KUKA KRL program: f1_Kuka_APT208T02S08.SRC

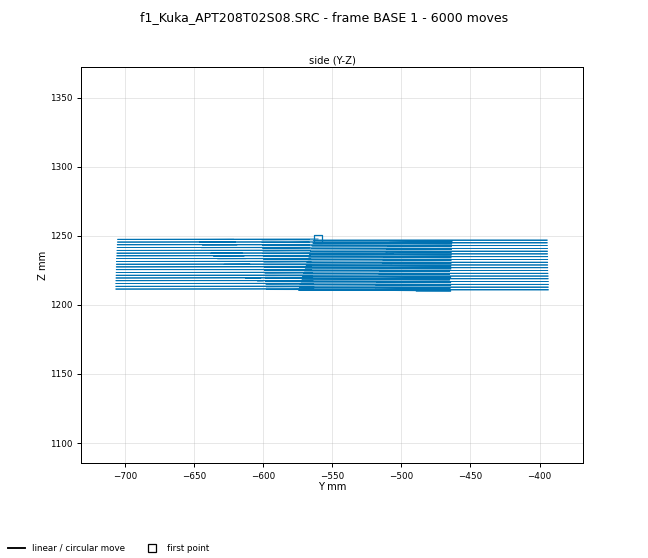
[picture p0: tool path of f1_Kuka_APT208T02S08.SRC in frame BASE 1, 6000 of 6001 moves have a stored position in this frame; points joined in program order, loops and branches not executed]
&ACCESS RVP
&REL 2
&PARAM TEMPLATE = C:\KRC\Roboter\Template\vorgabe
&PARAM EDITMASK = *
DEF f1_Kuka_APT208T02S08()


;FOLD INI;%{PE}%V3.2.0,%MKUKATPBASIS,%CINIT,%VCOMMON,%P
  ;FOLD BAS INI;%{E}%V3.2.0,%MKUKATPBASIS,%CINIT,%VINIT,%P
    GLOBAL INTERRUPT DECL 3 WHEN $STOPMESS==TRUE DO IR_STOPM ( )
    INTERRUPT ON 3
    BAS (#INITMOV,0 )
  ;ENDFOLD (BAS INI)
  ;FOLD USER INI;%{E}%V3.2.0,%MKUKATPUSER,%CINIT,%VINIT,%P
    ;Make your modifications here
  ;ENDFOLD (USER INI)
;ENDFOLD (INI)


;*** Make Null PTP Move
  PTP $pos_act

;*** Auto Load The Correct TOOL Data
  $tool=tool_data[2]

;*** Auto Load The Correct BASE Data
  $base=base_data[1]

  $ADVANCE = 5

;*** Restate Last Velocity
MMPM(30000.0)
SetRPM(8000)
LIN {X -0.044,Y -560.210,Z 1247.711,A 0.000,B 0.000,C 90.000,E1 163.921} C_DIS
LIN {X 0.207,Y -563.468,Z 1247.701,A 0.000,B 0.000,C 90.000,E1 162.236} C_DIS
LIN {X 0.002,Y -567.714,Z 1247.692,A 0.000,B 0.000,C 90.000,E1 160.604} C_DIS
LIN {X 0.261,Y -572.378,Z 1247.685,A 0.000,B 0.000,C 90.000,E1 159.209} C_DIS
LIN {X -0.101,Y -576.704,Z 1247.679,A 0.000,B 0.000,C 90.000,E1 158.156} C_DIS
LIN {X 0.147,Y -589.999,Z 1247.663,A 0.000,B 0.000,C 90.000,E1 155.305} C_DIS
LIN {X 0.135,Y -597.371,Z 1247.655,A 0.000,B 0.000,C 90.000,E1 153.845} C_DIS
LIN {X 0.131,Y -601.919,Z 1247.650,A 0.000,B 0.000,C 90.000,E1 152.922} C_DIS
LIN {X 0.032,Y -603.823,Z 1247.647,A 0.000,B 0.000,C 90.000,E1 152.538} C_DIS
LIN {X -0.143,Y -607.711,Z 1247.643,A 0.000,B 0.000,C 90.000,E1 151.769} C_DIS
LIN {X 0.008,Y -611.290,Z 1247.639,A 0.000,B 0.000,C 90.000,E1 150.973} C_DIS
LIN {X 0.120,Y -618.388,Z 1247.630,A 0.000,B 0.000,C 90.000,E1 149.410} C_DIS
LIN {X 0.147,Y -625.351,Z 1247.622,A 0.000,B 0.000,C 90.000,E1 147.867} C_DIS
LIN {X -0.054,Y -628.614,Z 1247.617,A 0.000,B 0.000,C 90.000,E1 147.120} C_DIS
LIN {X -0.384,Y -633.789,Z 1247.610,A 0.000,B 0.000,C 90.000,E1 145.881} C_DIS
LIN {X -0.147,Y -636.719,Z 1247.606,A 0.000,B 0.000,C 90.000,E1 145.102} C_DIS
LIN {X 0.026,Y -641.252,Z 1247.599,A 0.000,B 0.000,C 90.000,E1 143.829} C_DIS
LIN {X 0.272,Y -645.228,Z 1247.592,A 0.000,B 0.000,C 90.000,E1 142.557} C_DIS
LIN {X -0.366,Y -648.122,Z 1247.587,A 0.000,B 0.000,C 90.000,E1 141.618} C_DIS
LIN {X -0.126,Y -651.565,Z 1247.580,A 0.000,B 0.000,C 90.000,E1 140.356} C_DIS
LIN {X 0.124,Y -655.386,Z 1247.572,A 0.000,B 0.000,C 90.000,E1 138.852} C_DIS
LIN {X 0.020,Y -657.887,Z 1247.566,A 0.000,B 0.000,C 90.000,E1 137.877} C_DIS
LIN {X 0.341,Y -661.423,Z 1247.558,A 0.000,B 0.000,C 90.000,E1 136.377} C_DIS
LIN {X 0.254,Y -667.065,Z 1247.546,A 0.000,B 0.000,C 90.000,E1 134.190} C_DIS
LIN {X -0.167,Y -671.614,Z 1247.536,A 0.000,B 0.000,C 90.000,E1 132.528} C_DIS
LIN {X -0.020,Y -675.508,Z 1247.528,A 0.000,B 0.000,C 90.000,E1 131.067} C_DIS
LIN {X 0.168,Y -678.705,Z 1247.521,A 0.000,B 0.000,C 90.000,E1 129.850} C_DIS
LIN {X 0.172,Y -683.657,Z 1247.511,A 0.000,B 0.000,C 90.000,E1 127.935} C_DIS
LIN {X 0.214,Y -687.311,Z 1247.503,A 0.000,B 0.000,C 90.000,E1 126.503} C_DIS
LIN {X -0.308,Y -689.569,Z 1247.498,A 0.000,B 0.000,C 90.000,E1 125.598} C_DIS
LIN {X -0.197,Y -692.243,Z 1247.491,A 0.000,B 0.000,C 90.000,E1 124.405} C_DIS
LIN {X -0.081,Y -694.262,Z 1247.486,A 0.000,B 0.000,C 90.000,E1 123.452} C_DIS
LIN {X 0.093,Y -696.685,Z 1247.479,A 0.000,B 0.000,C 90.000,E1 122.260} C_DIS
LIN {X 0.151,Y -698.904,Z 1247.473,A 0.000,B 0.000,C 90.000,E1 121.082} C_DIS
LIN {X 0.008,Y -701.036,Z 1247.466,A 0.000,B 0.000,C 90.000,E1 119.922} C_DIS
LIN {X 0.209,Y -702.176,Z 1247.462,A 0.000,B 0.000,C 90.000,E1 119.205} C_DIS
LIN {X 0.084,Y -703.477,Z 1247.457,A 0.000,B 0.000,C 90.000,E1 118.281} C_DIS
LIN {X -0.359,Y -704.484,Z 1247.452,A 0.000,B 0.000,C 90.000,E1 117.385} C_DIS
LIN {X -0.127,Y -705.034,Z 1247.448,A 0.000,B 0.000,C 90.000,E1 116.668} C_DIS
LIN {X -0.206,Y -705.331,Z 1247.444,A 0.000,B 0.000,C 90.000,E1 115.976} C_DIS
LIN {X 0.373,Y -705.331,Z 1247.442,A 0.000,B 0.000,C 90.000,E1 115.463} C_DIS
LIN {X 0.013,Y -705.151,Z 1247.439,A 0.000,B 0.000,C 90.000,E1 115.027} C_DIS
LIN {X -0.052,Y -704.772,Z 1247.437,A 0.000,B 0.000,C 90.000,E1 114.567} C_DIS
LIN {X 0.229,Y -703.978,Z 1247.434,A 0.000,B 0.000,C 90.000,E1 114.079} C_DIS
LIN {X -0.131,Y -703.306,Z 1247.433,A 0.000,B 0.000,C 90.000,E1 113.875} C_DIS
LIN {X 0.144,Y -701.285,Z 1247.430,A 0.000,B 0.000,C 90.000,E1 113.387} C_DIS
LIN {X 0.280,Y -700.576,Z 1247.429,A 0.000,B 0.000,C 90.000,E1 113.259} C_DIS
LIN {X -0.106,Y -696.209,Z 1247.427,A 0.000,B 0.000,C 90.000,E1 112.823} C_DIS
LIN {X 0.023,Y -694.918,Z 1247.426,A 0.000,B 0.000,C 90.000,E1 112.695} C_DIS
LIN {X -0.059,Y -692.962,Z 1247.426,A 0.000,B 0.000,C 90.000,E1 112.589} C_DIS
LIN {X 0.208,Y -686.106,Z 1247.424,A 0.000,B 0.000,C 90.000,E1 112.333} C_DIS
LIN {X -0.047,Y -684.944,Z 1247.424,A 0.000,B 0.000,C 90.000,E1 112.333} C_DIS
LIN {X -0.092,Y -677.360,Z 1247.424,A 0.000,B 0.000,C 90.000,E1 112.259} C_DIS
LIN {X -0.131,Y -625.323,Z 1247.424,A 0.000,B 0.000,C 90.000,E1 112.259} C_DIS
LIN {X -0.005,Y -624.460,Z 1247.423,A 0.000,B 0.000,C 90.000,E1 112.206} C_DIS
LIN {X -0.259,Y -621.696,Z 1247.422,A 0.000,B 0.000,C 90.000,E1 112.025} C_DIS
LIN {X -0.295,Y -621.657,Z 1247.422,A 0.000,B 0.000,C 90.000,E1 112.025} C_DIS
LIN {X -0.018,Y -621.126,Z 1247.422,A 0.000,B 0.000,C 90.000,E1 111.897} C_DIS
LIN {X -0.061,Y -621.110,Z 1247.422,A 0.000,B 0.000,C 90.000,E1 111.897} C_DIS
LIN {X -0.234,Y -621.700,Z 1247.420,A 0.000,B 0.000,C 90.000,E1 111.589} C_DIS
LIN {X 0.091,Y -625.646,Z 1247.416,A 0.000,B 0.000,C 90.000,E1 110.791} C_DIS
LIN {X -0.347,Y -630.528,Z 1247.411,A 0.000,B 0.000,C 90.000,E1 109.939} C_DIS
LIN {X 0.056,Y -633.087,Z 1247.408,A 0.000,B 0.000,C 90.000,E1 109.396} C_DIS
LIN {X 0.311,Y -637.748,Z 1247.402,A 0.000,B 0.000,C 90.000,E1 108.362} C_DIS
LIN {X 0.156,Y -646.024,Z 1247.392,A 0.000,B 0.000,C 90.000,E1 106.622} C_DIS
LIN {X 0.043,Y -648.319,Z 1247.390,A 0.000,B 0.000,C 90.000,E1 106.134} C_DIS
LIN {X 0.257,Y -651.410,Z 1247.386,A 0.000,B 0.000,C 90.000,E1 105.371} C_DIS
LIN {X 0.003,Y -653.197,Z 1247.383,A 0.000,B 0.000,C 90.000,E1 104.898} C_DIS
LIN {X -0.197,Y -655.418,Z 1247.379,A 0.000,B 0.000,C 90.000,E1 104.175} C_DIS
LIN {X 0.208,Y -656.599,Z 1247.376,A 0.000,B 0.000,C 90.000,E1 103.647} C_DIS
LIN {X -0.126,Y -657.857,Z 1247.372,A 0.000,B 0.000,C 90.000,E1 102.939} C_DIS
LIN {X 0.298,Y -658.390,Z 1247.369,A 0.000,B 0.000,C 90.000,E1 102.411} C_DIS
LIN {X -0.054,Y -658.521,Z 1247.366,A 0.000,B 0.000,C 90.000,E1 101.951} C_DIS
LIN {X 0.273,Y -658.185,Z 1247.362,A 0.000,B 0.000,C 90.000,E1 101.186} C_DIS
LIN {X 0.054,Y -657.548,Z 1247.360,A 0.000,B 0.000,C 90.000,E1 100.715} C_DIS
LIN {X -0.290,Y -656.626,Z 1247.357,A 0.000,B 0.000,C 90.000,E1 100.254} C_DIS
LIN {X 0.124,Y -655.438,Z 1247.354,A 0.000,B 0.000,C 90.000,E1 99.726} C_DIS
LIN {X -0.105,Y -654.766,Z 1247.353,A 0.000,B 0.000,C 90.000,E1 99.500} C_DIS
LIN {X 0.293,Y -653.009,Z 1247.350,A 0.000,B 0.000,C 90.000,E1 98.973} C_DIS
LIN {X -0.070,Y -650.852,Z 1247.347,A 0.000,B 0.000,C 90.000,E1 98.511} C_DIS
LIN {X 0.171,Y -647.758,Z 1247.344,A 0.000,B 0.000,C 90.000,E1 97.871} C_DIS
LIN {X 0.294,Y -644.050,Z 1247.340,A 0.000,B 0.000,C 90.000,E1 97.239} C_DIS
LIN {X -0.248,Y -639.738,Z 1247.337,A 0.000,B 0.000,C 90.000,E1 96.663} C_DIS
LIN {X 0.077,Y -636.974,Z 1247.335,A 0.000,B 0.000,C 90.000,E1 96.258} C_DIS
LIN {X 0.143,Y -631.622,Z 1247.331,A 0.000,B 0.000,C 90.000,E1 95.625} C_DIS
LIN {X -0.307,Y -626.824,Z 1247.329,A 0.000,B 0.000,C 90.000,E1 95.163} C_DIS
LIN {X -0.030,Y -620.264,Z 1247.325,A 0.000,B 0.000,C 90.000,E1 94.531} C_DIS
LIN {X -0.028,Y -614.926,Z 1247.323,A 0.000,B 0.000,C 90.000,E1 94.073} C_DIS
LIN {X 0.146,Y -609.256,Z 1247.320,A 0.000,B 0.000,C 90.000,E1 93.612} C_DIS
LIN {X 0.021,Y -601.636,Z 1247.317,A 0.000,B 0.000,C 90.000,E1 93.094} C_DIS
LIN {X 0.005,Y -595.380,Z 1247.315,A 0.000,B 0.000,C 90.000,E1 92.694} C_DIS
LIN {X 0.222,Y -588.941,Z 1247.313,A 0.000,B 0.000,C 90.000,E1 92.293} C_DIS
LIN {X 0.267,Y -582.256,Z 1247.311,A 0.000,B 0.000,C 90.000,E1 91.949} C_DIS
LIN {X 0.028,Y -571.609,Z 1247.309,A 0.000,B 0.000,C 90.000,E1 91.547} C_DIS
LIN {X -0.094,Y -570.151,Z 1247.308,A 0.000,B 0.000,C 90.000,E1 91.489} C_DIS
LIN {X -0.132,Y -568.129,Z 1247.308,A 0.000,B 0.000,C 90.000,E1 91.375} C_DIS
LIN {X -0.189,Y -568.057,Z 1247.308,A 0.000,B 0.000,C 90.000,E1 91.375} C_DIS
LIN {X 0.032,Y -566.808,Z 1247.306,A 0.000,B 0.000,C 90.000,E1 91.088} C_DIS
LIN {X -0.010,Y -566.801,Z 1247.306,A 0.000,B 0.000,C 90.000,E1 91.088} C_DIS
LIN {X 0.198,Y -566.625,Z 1247.304,A 0.000,B 0.000,C 90.000,E1 90.630} C_DIS
LIN {X -0.016,Y -567.066,Z 1247.299,A 0.000,B 0.000,C 90.000,E1 89.828} C_DIS
LIN {X 0.153,Y -568.269,Z 1247.290,A 0.000,B 0.000,C 90.000,E1 88.165} C_DIS
LIN {X 0.024,Y -570.020,Z 1247.278,A 0.000,B 0.000,C 90.000,E1 85.988} C_DIS
LIN {X -0.118,Y -571.911,Z 1247.267,A 0.000,B 0.000,C 90.000,E1 84.090} C_DIS
LIN {X 0.298,Y -573.564,Z 1247.258,A 0.000,B 0.000,C 90.000,E1 82.413} C_DIS
LIN {X -0.014,Y -574.966,Z 1247.250,A 0.000,B 0.000,C 90.000,E1 81.084} C_DIS
LIN {X 0.143,Y -575.994,Z 1247.245,A 0.000,B 0.000,C 90.000,E1 79.982} C_DIS
LIN {X 0.064,Y -577.006,Z 1247.237,A 0.000,B 0.000,C 90.000,E1 78.634} C_DIS
LIN {X 0.014,Y -577.979,Z 1247.229,A 0.000,B 0.000,C 90.000,E1 77.285} C_DIS
LIN {X 0.102,Y -578.547,Z 1247.225,A 0.000,B 0.000,C 90.000,E1 76.464} C_DIS
LIN {X 0.211,Y -579.429,Z 1247.217,A 0.000,B 0.000,C 90.000,E1 75.102} C_DIS
LIN {X -0.011,Y -580.339,Z 1247.208,A 0.000,B 0.000,C 90.000,E1 73.504} C_DIS
LIN {X 0.115,Y -581.232,Z 1247.199,A 0.000,B 0.000,C 90.000,E1 71.873} C_DIS
LIN {X -0.131,Y -582.131,Z 1247.192,A 0.000,B 0.000,C 90.000,E1 70.550} C_DIS
LIN {X 0.140,Y -583.605,Z 1247.178,A 0.000,B 0.000,C 90.000,E1 68.103} C_DIS
LIN {X -0.050,Y -585.213,Z 1247.167,A 0.000,B 0.000,C 90.000,E1 65.973} C_DIS
LIN {X -0.250,Y -586.167,Z 1247.161,A 0.000,B 0.000,C 90.000,E1 64.921} C_DIS
LIN {X 0.016,Y -588.286,Z 1247.147,A 0.000,B 0.000,C 90.000,E1 62.487} C_DIS
LIN {X 0.143,Y -589.936,Z 1247.138,A 0.000,B 0.000,C 90.000,E1 60.873} C_DIS
LIN {X 0.181,Y -591.324,Z 1247.131,A 0.000,B 0.000,C 90.000,E1 59.537} C_DIS
LIN {X 0.249,Y -592.705,Z 1247.124,A 0.000,B 0.000,C 90.000,E1 58.201} C_DIS
LIN {X -0.166,Y -593.989,Z 1247.116,A 0.000,B 0.000,C 90.000,E1 56.914} C_DIS
LIN {X -0.010,Y -595.441,Z 1247.107,A 0.000,B 0.000,C 90.000,E1 55.308} C_DIS
LIN {X 0.179,Y -596.833,Z 1247.099,A 0.000,B 0.000,C 90.000,E1 53.703} C_DIS
LIN {X -0.336,Y -598.277,Z 1247.088,A 0.000,B 0.000,C 90.000,E1 51.904} C_DIS
LIN {X 0.142,Y -599.069,Z 1247.082,A 0.000,B 0.000,C 90.000,E1 50.803} C_DIS
LIN {X 0.189,Y -599.846,Z 1247.074,A 0.000,B 0.000,C 90.000,E1 49.218} C_DIS
LIN {X 0.229,Y -600.315,Z 1247.068,A 0.000,B 0.000,C 90.000,E1 48.162} C_DIS
LIN {X 0.037,Y -600.654,Z 1247.063,A 0.000,B 0.000,C 90.000,E1 47.391} C_DIS
LIN {X 0.068,Y -600.929,Z 1247.055,A 0.000,B 0.000,C 90.000,E1 45.810} C_DIS
LIN {X 0.090,Y -600.994,Z 1247.049,A 0.000,B 0.000,C 90.000,E1 44.757} C_DIS
LIN {X 0.111,Y -600.833,Z 1247.043,A 0.000,B 0.000,C 90.000,E1 43.704} C_DIS
LIN {X -0.055,Y -600.482,Z 1247.036,A 0.000,B 0.000,C 90.000,E1 42.405} C_DIS
LIN {X -0.040,Y -599.793,Z 1247.027,A 0.000,B 0.000,C 90.000,E1 40.825} C_DIS
LIN {X 0.229,Y -599.080,Z 1247.020,A 0.000,B 0.000,C 90.000,E1 39.483} C_DIS
LIN {X -0.127,Y -598.295,Z 1247.014,A 0.000,B 0.000,C 90.000,E1 38.463} C_DIS
LIN {X 0.111,Y -597.624,Z 1247.009,A 0.000,B 0.000,C 90.000,E1 37.649} C_DIS
LIN {X 0.211,Y -596.519,Z 1247.003,A 0.000,B 0.000,C 90.000,E1 36.583} C_DIS
LIN {X 0.296,Y -595.048,Z 1246.998,A 0.000,B 0.000,C 90.000,E1 35.518} C_DIS
LIN {X 0.136,Y -593.782,Z 1246.993,A 0.000,B 0.000,C 90.000,E1 34.739} C_DIS
LIN {X -0.159,Y -591.802,Z 1246.987,A 0.000,B 0.000,C 90.000,E1 33.706} C_DIS
LIN {X 0.135,Y -590.025,Z 1246.983,A 0.000,B 0.000,C 90.000,E1 32.880} C_DIS
LIN {X 0.214,Y -588.683,Z 1246.980,A 0.000,B 0.000,C 90.000,E1 32.339} C_DIS
LIN {X 0.161,Y -586.395,Z 1246.975,A 0.000,B 0.000,C 90.000,E1 31.544} C_DIS
LIN {X 0.091,Y -583.801,Z 1246.971,A 0.000,B 0.000,C 90.000,E1 30.747} C_DIS
LIN {X -0.006,Y -580.713,Z 1246.966,A 0.000,B 0.000,C 90.000,E1 29.951} C_DIS
LIN {X 0.008,Y -578.463,Z 1246.964,A 0.000,B 0.000,C 90.000,E1 29.411} C_DIS
LIN {X 0.000,Y -575.979,Z 1246.960,A 0.000,B 0.000,C 90.000,E1 28.871} C_DIS
LIN {X 0.228,Y -571.161,Z 1246.955,A 0.000,B 0.000,C 90.000,E1 27.897} C_DIS
LIN {X -0.280,Y -566.486,Z 1246.951,A 0.000,B 0.000,C 90.000,E1 27.129} C_DIS
LIN {X 0.116,Y -563.139,Z 1246.948,A 0.000,B 0.000,C 90.000,E1 26.539} C_DIS
LIN {X 0.233,Y -559.571,Z 1246.944,A 0.000,B 0.000,C 90.000,E1 25.976} C_DIS
LIN {X -0.175,Y -555.773,Z 1246.941,A 0.000,B 0.000,C 90.000,E1 25.463} C_DIS
LIN {X -0.105,Y -551.668,Z 1246.938,A 0.000,B 0.000,C 90.000,E1 24.899} C_DIS
LIN {X 0.196,Y -545.099,Z 1246.934,A 0.000,B 0.000,C 90.000,E1 24.027} C_DIS
LIN {X 0.123,Y -539.158,Z 1246.930,A 0.000,B 0.000,C 90.000,E1 23.334} C_DIS
LIN {X -0.172,Y -531.578,Z 1246.925,A 0.000,B 0.000,C 90.000,E1 22.514} C_DIS
LIN {X 0.065,Y -524.997,Z 1246.921,A 0.000,B 0.000,C 90.000,E1 21.791} C_DIS
LIN {X -0.124,Y -515.656,Z 1246.916,A 0.000,B 0.000,C 90.000,E1 20.844} C_DIS
LIN {X 0.061,Y -507.377,Z 1246.911,A 0.000,B 0.000,C 90.000,E1 19.993} C_DIS
LIN {X -0.230,Y -497.632,Z 1246.906,A 0.000,B 0.000,C 90.000,E1 19.087} C_DIS
LIN {X -0.071,Y -487.541,Z 1246.901,A 0.000,B 0.000,C 90.000,E1 18.127} C_DIS
LIN {X -0.049,Y -478.666,Z 1246.896,A 0.000,B 0.000,C 90.000,E1 17.330} C_DIS
LIN {X -0.150,Y -462.368,Z 1246.888,A 0.000,B 0.000,C 90.000,E1 15.898} C_DIS
LIN {X -0.017,Y -446.234,Z 1246.880,A 0.000,B 0.000,C 90.000,E1 14.411} C_DIS
LIN {X 0.099,Y -424.423,Z 1246.868,A 0.000,B 0.000,C 90.000,E1 12.243} C_DIS
LIN {X -0.111,Y -405.887,Z 1246.857,A 0.000,B 0.000,C 90.000,E1 10.254} C_DIS
LIN {X -0.165,Y -401.633,Z 1246.854,A 0.000,B 0.000,C 90.000,E1 9.782} C_DIS
LIN {X 0.209,Y -396.128,Z 1246.850,A 0.000,B 0.000,C 90.000,E1 8.973} C_DIS
LIN {X 0.139,Y -394.399,Z 1246.848,A 0.000,B 0.000,C 90.000,E1 8.624} C_DIS
LIN {X 0.103,Y -394.392,Z 1246.848,A 0.000,B 0.000,C 90.000,E1 8.624} C_DIS
LIN {X -0.056,Y -394.298,Z 1246.848,A 0.000,B 0.000,C 90.000,E1 8.568} C_DIS
LIN {X -0.092,Y -394.300,Z 1246.848,A 0.000,B 0.000,C 90.000,E1 8.568} C_DIS
LIN {X -0.043,Y -396.382,Z 1246.845,A 0.000,B 0.000,C 90.000,E1 8.106} C_DIS
LIN {X 0.065,Y -400.030,Z 1246.843,A 0.000,B 0.000,C 90.000,E1 7.701} C_DIS
LIN {X -0.161,Y -405.750,Z 1246.840,A 0.000,B 0.000,C 90.000,E1 7.296} C_DIS
LIN {X -0.113,Y -412.470,Z 1246.838,A 0.000,B 0.000,C 90.000,E1 6.834} C_DIS
LIN {X -0.049,Y -423.583,Z 1246.833,A 0.000,B 0.000,C 90.000,E1 6.030} C_DIS
LIN {X -0.118,Y -431.436,Z 1246.830,A 0.000,B 0.000,C 90.000,E1 5.448} C_DIS
LIN {X -0.078,Y -440.778,Z 1246.826,A 0.000,B 0.000,C 90.000,E1 4.702} C_DIS
LIN {X -0.019,Y -448.647,Z 1246.823,A 0.000,B 0.000,C 90.000,E1 4.073} C_DIS
LIN {X -0.185,Y -459.503,Z 1246.818,A 0.000,B 0.000,C 90.000,E1 3.212} C_DIS
LIN {X -0.227,Y -467.080,Z 1246.814,A 0.000,B 0.000,C 90.000,E1 2.579} C_DIS
LIN {X 0.174,Y -472.961,Z 1246.811,A 0.000,B 0.000,C 90.000,E1 2.007} C_DIS
LIN {X -0.051,Y -478.704,Z 1246.808,A 0.000,B 0.000,C 90.000,E1 1.489} C_DIS
LIN {X -0.207,Y -485.431,Z 1246.804,A 0.000,B 0.000,C 90.000,E1 0.802} C_DIS
LIN {X 0.000,Y -492.261,Z 1246.800,A 0.000,B 0.000,C 90.000,E1 360.000} C_DIS
LIN {X 0.038,Y -496.537,Z 1246.797,A 0.000,B 0.000,C 90.000,E1 359.484} C_DIS
LIN {X 0.141,Y -503.300,Z 1246.792,A 0.000,B 0.000,C 90.000,E1 358.568} C_DIS
LIN {X -0.071,Y -507.579,Z 1246.789,A 0.000,B 0.000,C 90.000,E1 357.993} C_DIS
LIN {X -0.058,Y -512.453,Z 1246.785,A 0.000,B 0.000,C 90.000,E1 357.249} C_DIS
LIN {X 0.021,Y -517.080,Z 1246.781,A 0.000,B 0.000,C 90.000,E1 356.502} C_DIS
LIN {X -0.081,Y -520.544,Z 1246.777,A 0.000,B 0.000,C 90.000,E1 355.927} C_DIS
LIN {X 0.080,Y -524.508,Z 1246.773,A 0.000,B 0.000,C 90.000,E1 355.179} C_DIS
LIN {X 0.279,Y -528.131,Z 1246.769,A 0.000,B 0.000,C 90.000,E1 354.432} C_DIS
LIN {X 0.261,Y -530.849,Z 1246.766,A 0.000,B 0.000,C 90.000,E1 353.856} C_DIS
LIN {X 0.262,Y -533.398,Z 1246.763,A 0.000,B 0.000,C 90.000,E1 353.280} C_DIS
LIN {X -0.254,Y -535.770,Z 1246.760,A 0.000,B 0.000,C 90.000,E1 352.761} C_DIS
LIN {X -0.170,Y -538.958,Z 1246.755,A 0.000,B 0.000,C 90.000,E1 351.894} C_DIS
LIN {X 0.021,Y -542.828,Z 1246.749,A 0.000,B 0.000,C 90.000,E1 350.735} C_DIS
LIN {X 0.270,Y -545.377,Z 1246.744,A 0.000,B 0.000,C 90.000,E1 349.859} C_DIS
LIN {X 0.012,Y -548.535,Z 1246.738,A 0.000,B 0.000,C 90.000,E1 348.757} C_DIS
LIN {X -0.212,Y -550.682,Z 1246.733,A 0.000,B 0.000,C 90.000,E1 347.937} C_DIS
LIN {X -0.299,Y -553.228,Z 1246.727,A 0.000,B 0.000,C 90.000,E1 346.825} C_DIS
LIN {X -0.221,Y -555.597,Z 1246.720,A 0.000,B 0.000,C 90.000,E1 345.700} C_DIS
LIN {X -0.237,Y -557.140,Z 1246.716,A 0.000,B 0.000,C 90.000,E1 344.866} C_DIS
LIN {X -0.100,Y -559.042,Z 1246.710,A 0.000,B 0.000,C 90.000,E1 343.740} C_DIS
LIN {X -0.080,Y -560.216,Z 1246.705,A 0.000,B 0.000,C 90.000,E1 342.906} C_DIS
LIN {X -0.278,Y -561.613,Z 1246.699,A 0.000,B 0.000,C 90.000,E1 341.819} C_DIS
LIN {X 0.074,Y -562.633,Z 1246.693,A 0.000,B 0.000,C 90.000,E1 340.678} C_DIS
LIN {X -0.225,Y -563.146,Z 1246.688,A 0.000,B 0.000,C 90.000,E1 339.880} C_DIS
LIN {X 0.012,Y -563.378,Z 1246.684,A 0.000,B 0.000,C 90.000,E1 339.028} C_DIS
LIN {X 0.131,Y -563.407,Z 1246.681,A 0.000,B 0.000,C 90.000,E1 338.465} C_DIS
LIN {X -0.155,Y -563.100,Z 1246.676,A 0.000,B 0.000,C 90.000,E1 337.667} C_DIS
LIN {X -0.032,Y -562.690,Z 1246.673,A 0.000,B 0.000,C 90.000,E1 337.102} C_DIS
LIN {X -0.018,Y -561.489,Z 1246.667,A 0.000,B 0.000,C 90.000,E1 335.997} C_DIS
LIN {X 0.092,Y -560.672,Z 1246.664,A 0.000,B 0.000,C 90.000,E1 335.433} C_DIS
LIN {X 0.232,Y -559.167,Z 1246.659,A 0.000,B 0.000,C 90.000,E1 334.588} C_DIS
LIN {X -0.299,Y -556.141,Z 1246.651,A 0.000,B 0.000,C 90.000,E1 333.256} C_DIS
LIN {X -0.193,Y -553.609,Z 1246.647,A 0.000,B 0.000,C 90.000,E1 332.410} C_DIS
LIN {X -0.113,Y -550.710,Z 1246.642,A 0.000,B 0.000,C 90.000,E1 331.563} C_DIS
LIN {X 0.054,Y -547.836,Z 1246.638,A 0.000,B 0.000,C 90.000,E1 330.845} C_DIS
LIN {X 0.189,Y -544.503,Z 1246.634,A 0.000,B 0.000,C 90.000,E1 330.127} C_DIS
LIN {X -0.180,Y -540.698,Z 1246.630,A 0.000,B 0.000,C 90.000,E1 329.459} C_DIS
LIN {X 0.023,Y -535.345,Z 1246.625,A 0.000,B 0.000,C 90.000,E1 328.584} C_DIS
LIN {X 0.013,Y -528.671,Z 1246.620,A 0.000,B 0.000,C 90.000,E1 327.582} C_DIS
LIN {X 0.073,Y -522.477,Z 1246.615,A 0.000,B 0.000,C 90.000,E1 326.707} C_DIS
LIN {X -0.080,Y -516.644,Z 1246.610,A 0.000,B 0.000,C 90.000,E1 325.881} C_DIS
LIN {X 0.194,Y -513.232,Z 1246.607,A 0.000,B 0.000,C 90.000,E1 325.308} C_DIS
LIN {X 0.218,Y -510.256,Z 1246.604,A 0.000,B 0.000,C 90.000,E1 324.769} C_DIS
LIN {X -0.293,Y -507.821,Z 1246.601,A 0.000,B 0.000,C 90.000,E1 324.196} C_DIS
LIN {X 0.126,Y -506.615,Z 1246.599,A 0.000,B 0.000,C 90.000,E1 323.703} C_DIS
LIN {X -0.173,Y -504.975,Z 1246.594,A 0.000,B 0.000,C 90.000,E1 322.844} C_DIS
LIN {X 0.217,Y -504.261,Z 1246.589,A 0.000,B 0.000,C 90.000,E1 321.904} C_DIS
LIN {X -0.112,Y -504.155,Z 1246.584,A 0.000,B 0.000,C 90.000,E1 321.045} C_DIS
LIN {X 0.179,Y -504.992,Z 1246.569,A 0.000,B 0.000,C 90.000,E1 318.324} C_DIS
LIN {X -0.015,Y -505.613,Z 1246.557,A 0.000,B 0.000,C 90.000,E1 316.257} C_DIS
LIN {X -0.165,Y -505.927,Z 1246.550,A 0.000,B 0.000,C 90.000,E1 315.081} C_DIS
LIN {X 0.153,Y -506.372,Z 1246.540,A 0.000,B 0.000,C 90.000,E1 313.257} C_DIS
LIN {X 0.016,Y -506.745,Z 1246.534,A 0.000,B 0.000,C 90.000,E1 312.081} C_DIS
LIN {X -0.002,Y -507.285,Z 1246.524,A 0.000,B 0.000,C 90.000,E1 310.297} C_DIS
LIN {X -0.083,Y -507.528,Z 1246.517,A 0.000,B 0.000,C 90.000,E1 309.116} C_DIS
LIN {X 0.050,Y -508.042,Z 1246.507,A 0.000,B 0.000,C 90.000,E1 307.317} C_DIS
LIN {X -0.026,Y -508.356,Z 1246.501,A 0.000,B 0.000,C 90.000,E1 306.137} C_DIS
LIN {X -0.090,Y -508.583,Z 1246.493,A 0.000,B 0.000,C 90.000,E1 304.659} C_DIS
LIN {X -0.013,Y -508.797,Z 1246.484,A 0.000,B 0.000,C 90.000,E1 303.166} C_DIS
LIN {X 0.075,Y -508.907,Z 1246.476,A 0.000,B 0.000,C 90.000,E1 301.671} C_DIS
LIN {X -0.134,Y -508.877,Z 1246.464,A 0.000,B 0.000,C 90.000,E1 299.617} C_DIS
LIN {X 0.046,Y -508.833,Z 1246.458,A 0.000,B 0.000,C 90.000,E1 298.409} C_DIS
LIN {X 0.058,Y -508.718,Z 1246.450,A 0.000,B 0.000,C 90.000,E1 296.924} C_DIS
LIN {X -0.111,Y -508.723,Z 1246.437,A 0.000,B 0.000,C 90.000,E1 294.567} C_DIS
LIN {X 0.089,Y -508.797,Z 1246.433,A 0.000,B 0.000,C 90.000,E1 293.951} C_DIS
LIN {X 0.136,Y -508.606,Z 1246.425,A 0.000,B 0.000,C 90.000,E1 292.461} C_DIS
LIN {X -0.027,Y -508.324,Z 1246.420,A 0.000,B 0.000,C 90.000,E1 291.589} C_DIS
LIN {X -0.179,Y -507.655,Z 1246.412,A 0.000,B 0.000,C 90.000,E1 290.120} C_DIS
LIN {X 0.156,Y -506.724,Z 1246.400,A 0.000,B 0.000,C 90.000,E1 288.000} C_DIS
LIN {X 0.204,Y -506.342,Z 1246.394,A 0.000,B 0.000,C 90.000,E1 286.804} C_DIS
LIN {X 0.188,Y -505.727,Z 1246.385,A 0.000,B 0.000,C 90.000,E1 285.315} C_DIS
LIN {X 0.158,Y -504.856,Z 1246.377,A 0.000,B 0.000,C 90.000,E1 283.828} C_DIS
LIN {X -0.080,Y -503.616,Z 1246.367,A 0.000,B 0.000,C 90.000,E1 282.063} C_DIS
LIN {X 0.043,Y -502.285,Z 1246.357,A 0.000,B 0.000,C 90.000,E1 280.254} C_DIS
LIN {X 0.121,Y -501.261,Z 1246.349,A 0.000,B 0.000,C 90.000,E1 278.746} C_DIS
LIN {X -0.259,Y -499.624,Z 1246.334,A 0.000,B 0.000,C 90.000,E1 276.087} C_DIS
LIN {X 0.198,Y -498.885,Z 1246.325,A 0.000,B 0.000,C 90.000,E1 274.531} C_DIS
LIN {X -0.041,Y -497.836,Z 1246.315,A 0.000,B 0.000,C 90.000,E1 272.751} C_DIS
LIN {X -0.058,Y -496.883,Z 1246.309,A 0.000,B 0.000,C 90.000,E1 271.547} C_DIS
LIN {X -0.157,Y -495.147,Z 1246.295,A 0.000,B 0.000,C 90.000,E1 269.141} C_DIS
LIN {X -0.008,Y -493.925,Z 1246.285,A 0.000,B 0.000,C 90.000,E1 267.306} C_DIS
LIN {X -0.155,Y -493.819,Z 1246.283,A 0.000,B 0.000,C 90.000,E1 267.020} C_DIS
LIN {X -0.200,Y -493.064,Z 1246.277,A 0.000,B 0.000,C 90.000,E1 265.812} C_DIS
LIN {X 0.086,Y -492.259,Z 1246.268,A 0.000,B 0.000,C 90.000,E1 264.261} C_DIS
LIN {X -0.090,Y -491.179,Z 1246.260,A 0.000,B 0.000,C 90.000,E1 262.761} C_DIS
LIN {X 0.264,Y -489.818,Z 1246.251,A 0.000,B 0.000,C 90.000,E1 261.197} C_DIS
LIN {X -0.241,Y -487.525,Z 1246.238,A 0.000,B 0.000,C 90.000,E1 258.814} C_DIS
LIN {X 0.098,Y -486.156,Z 1246.228,A 0.000,B 0.000,C 90.000,E1 256.937} C_DIS
LIN {X 0.051,Y -485.013,Z 1246.217,A 0.000,B 0.000,C 90.000,E1 255.102} C_DIS
LIN {X 0.110,Y -484.152,Z 1246.209,A 0.000,B 0.000,C 90.000,E1 253.559} C_DIS
LIN {X 0.134,Y -482.924,Z 1246.197,A 0.000,B 0.000,C 90.000,E1 251.402} C_DIS
LIN {X -0.022,Y -481.965,Z 1246.187,A 0.000,B 0.000,C 90.000,E1 249.571} C_DIS
LIN {X -0.020,Y -481.180,Z 1246.178,A 0.000,B 0.000,C 90.000,E1 248.028} C_DIS
LIN {X -0.043,Y -480.072,Z 1246.168,A 0.000,B 0.000,C 90.000,E1 246.177} C_DIS
LIN {X 0.098,Y -478.960,Z 1246.159,A 0.000,B 0.000,C 90.000,E1 244.613} C_DIS
LIN {X -0.011,Y -477.875,Z 1246.151,A 0.000,B 0.000,C 90.000,E1 243.076} C_DIS
LIN {X -0.111,Y -476.970,Z 1246.144,A 0.000,B 0.000,C 90.000,E1 241.847} C_DIS
LIN {X 0.198,Y -475.709,Z 1246.135,A 0.000,B 0.000,C 90.000,E1 240.255} C_DIS
LIN {X 0.302,Y -474.600,Z 1246.128,A 0.000,B 0.000,C 90.000,E1 238.997} C_DIS
LIN {X 0.116,Y -472.593,Z 1246.116,A 0.000,B 0.000,C 90.000,E1 236.834} C_DIS
LIN {X -0.259,Y -470.759,Z 1246.104,A 0.000,B 0.000,C 90.000,E1 234.689} C_DIS
LIN {X 0.067,Y -468.783,Z 1246.088,A 0.000,B 0.000,C 90.000,E1 231.823} C_DIS
LIN {X -0.137,Y -467.697,Z 1246.079,A 0.000,B 0.000,C 90.000,E1 230.275} C_DIS
LIN {X -0.061,Y -466.646,Z 1246.071,A 0.000,B 0.000,C 90.000,E1 228.690} C_DIS
LIN {X 0.111,Y -465.092,Z 1246.058,A 0.000,B 0.000,C 90.000,E1 226.458} C_DIS
LIN {X -0.038,Y -463.157,Z 1246.034,A 0.000,B 0.000,C 90.000,E1 222.043} C_DIS
LIN {X 0.013,Y -464.466,Z 1246.000,A 0.000,B 0.000,C 90.000,E1 216.011} C_DIS
LIN {X -0.043,Y -467.702,Z 1245.976,A 0.000,B 0.000,C 90.000,E1 211.592} C_DIS
LIN {X -0.220,Y -470.018,Z 1245.963,A 0.000,B 0.000,C 90.000,E1 209.411} C_DIS
LIN {X 0.025,Y -473.166,Z 1245.949,A 0.000,B 0.000,C 90.000,E1 206.873} C_DIS
LIN {X 0.034,Y -478.126,Z 1245.929,A 0.000,B 0.000,C 90.000,E1 203.131} C_DIS
LIN {X -0.216,Y -483.876,Z 1245.910,A 0.000,B 0.000,C 90.000,E1 199.758} C_DIS
LIN {X 0.009,Y -488.813,Z 1245.896,A 0.000,B 0.000,C 90.000,E1 197.275} C_DIS
LIN {X 0.177,Y -492.910,Z 1245.886,A 0.000,B 0.000,C 90.000,E1 195.426} C_DIS
LIN {X -0.173,Y -497.099,Z 1245.876,A 0.000,B 0.000,C 90.000,E1 193.647} C_DIS
LIN {X 0.217,Y -503.520,Z 1245.861,A 0.000,B 0.000,C 90.000,E1 190.894} C_DIS
LIN {X -0.215,Y -508.030,Z 1245.851,A 0.000,B 0.000,C 90.000,E1 189.151} C_DIS
LIN {X -0.049,Y -512.595,Z 1245.841,A 0.000,B 0.000,C 90.000,E1 187.352} C_DIS
LIN {X 0.170,Y -516.376,Z 1245.833,A 0.000,B 0.000,C 90.000,E1 185.853} C_DIS
LIN {X -0.166,Y -520.846,Z 1245.823,A 0.000,B 0.000,C 90.000,E1 184.131} C_DIS
LIN {X 0.161,Y -524.533,Z 1245.815,A 0.000,B 0.000,C 90.000,E1 182.636} C_DIS
LIN {X -0.026,Y -528.869,Z 1245.805,A 0.000,B 0.000,C 90.000,E1 180.917} C_DIS
LIN {X -0.130,Y -533.101,Z 1245.796,A 0.000,B 0.000,C 90.000,E1 179.198} C_DIS
LIN {X -0.137,Y -535.872,Z 1245.789,A 0.000,B 0.000,C 90.000,E1 178.051} C_DIS
LIN {X -0.088,Y -539.072,Z 1245.781,A 0.000,B 0.000,C 90.000,E1 176.617} C_DIS
LIN {X -0.007,Y -541.504,Z 1245.775,A 0.000,B 0.000,C 90.000,E1 175.469} C_DIS
LIN {X 0.168,Y -544.420,Z 1245.767,A 0.000,B 0.000,C 90.000,E1 174.033} C_DIS
LIN {X -0.092,Y -547.170,Z 1245.759,A 0.000,B 0.000,C 90.000,E1 172.648} C_DIS
LIN {X 0.217,Y -549.283,Z 1245.753,A 0.000,B 0.000,C 90.000,E1 171.489} C_DIS
LIN {X 0.242,Y -552.243,Z 1245.744,A 0.000,B 0.000,C 90.000,E1 169.803} C_DIS
LIN {X 0.199,Y -554.593,Z 1245.736,A 0.000,B 0.000,C 90.000,E1 168.409} C_DIS
LIN {X 0.014,Y -557.300,Z 1245.726,A 0.000,B 0.000,C 90.000,E1 166.756} C_DIS
LIN {X 0.181,Y -560.991,Z 1245.714,A 0.000,B 0.000,C 90.000,E1 164.519} C_DIS
LIN {X 0.203,Y -565.306,Z 1245.702,A 0.000,B 0.000,C 90.000,E1 162.308} C_DIS
LIN {X 0.027,Y -569.626,Z 1245.693,A 0.000,B 0.000,C 90.000,E1 160.678} C_DIS
LIN {X -0.225,Y -574.312,Z 1245.685,A 0.000,B 0.000,C 90.000,E1 159.337} C_DIS
LIN {X -0.029,Y -578.628,Z 1245.679,A 0.000,B 0.000,C 90.000,E1 158.230} C_DIS
LIN {X -0.022,Y -591.691,Z 1245.663,A 0.000,B 0.000,C 90.000,E1 155.409} C_DIS
LIN {X 0.008,Y -598.864,Z 1245.655,A 0.000,B 0.000,C 90.000,E1 153.948} C_DIS
LIN {X 0.262,Y -603.918,Z 1245.649,A 0.000,B 0.000,C 90.000,E1 152.871} C_DIS
LIN {X 0.037,Y -608.822,Z 1245.644,A 0.000,B 0.000,C 90.000,E1 151.847} C_DIS
LIN {X 0.157,Y -613.470,Z 1245.638,A 0.000,B 0.000,C 90.000,E1 150.795} C_DIS
LIN {X -0.215,Y -619.160,Z 1245.631,A 0.000,B 0.000,C 90.000,E1 149.537} C_DIS
LIN {X 0.053,Y -622.564,Z 1245.626,A 0.000,B 0.000,C 90.000,E1 148.742} C_DIS
LIN {X 0.155,Y -626.947,Z 1245.621,A 0.000,B 0.000,C 90.000,E1 147.709} C_DIS
LIN {X -0.026,Y -630.120,Z 1245.616,A 0.000,B 0.000,C 90.000,E1 146.962} C_DIS
LIN {X 0.202,Y -635.128,Z 1245.609,A 0.000,B 0.000,C 90.000,E1 145.674} C_DIS
LIN {X -0.434,Y -637.924,Z 1245.605,A 0.000,B 0.000,C 90.000,E1 144.975} C_DIS
LIN {X 0.247,Y -641.459,Z 1245.600,A 0.000,B 0.000,C 90.000,E1 143.909} C_DIS
LIN {X -0.332,Y -643.828,Z 1245.595,A 0.000,B 0.000,C 90.000,E1 143.210} C_DIS
LIN {X -0.083,Y -646.850,Z 1245.590,A 0.000,B 0.000,C 90.000,E1 142.190} C_DIS
LIN {X 0.140,Y -650.299,Z 1245.583,A 0.000,B 0.000,C 90.000,E1 140.928} C_DIS
LIN {X 0.004,Y -653.526,Z 1245.576,A 0.000,B 0.000,C 90.000,E1 139.703} C_DIS
LIN {X -0.168,Y -656.666,Z 1245.569,A 0.000,B 0.000,C 90.000,E1 138.485} C_DIS
LIN {X 0.182,Y -659.076,Z 1245.564,A 0.000,B 0.000,C 90.000,E1 137.472} C_DIS
LIN {X -0.419,Y -663.206,Z 1245.554,A 0.000,B 0.000,C 90.000,E1 135.810} C_DIS
LIN {X 0.020,Y -668.256,Z 1245.544,A 0.000,B 0.000,C 90.000,E1 133.824} C_DIS
LIN {X 0.071,Y -672.125,Z 1245.535,A 0.000,B 0.000,C 90.000,E1 132.366} C_DIS
LIN {X 0.207,Y -675.356,Z 1245.529,A 0.000,B 0.000,C 90.000,E1 131.148} C_DIS
LIN {X -0.013,Y -679.149,Z 1245.521,A 0.000,B 0.000,C 90.000,E1 129.725} C_DIS
LIN {X -0.022,Y -683.490,Z 1245.511,A 0.000,B 0.000,C 90.000,E1 128.051} C_DIS
LIN {X -0.109,Y -687.136,Z 1245.504,A 0.000,B 0.000,C 90.000,E1 126.629} C_DIS
LIN {X -0.080,Y -689.404,Z 1245.498,A 0.000,B 0.000,C 90.000,E1 125.678} C_DIS
LIN {X 0.034,Y -692.086,Z 1245.492,A 0.000,B 0.000,C 90.000,E1 124.485} C_DIS
LIN {X -0.427,Y -694.116,Z 1245.486,A 0.000,B 0.000,C 90.000,E1 123.579} C_DIS
LIN {X 0.329,Y -696.566,Z 1245.480,A 0.000,B 0.000,C 90.000,E1 122.339} C_DIS
LIN {X -0.208,Y -698.796,Z 1245.473,A 0.000,B 0.000,C 90.000,E1 121.209} C_DIS
LIN {X 0.252,Y -700.963,Z 1245.467,A 0.000,B 0.000,C 90.000,E1 120.001} C_DIS
LIN {X 0.116,Y -702.479,Z 1245.462,A 0.000,B 0.000,C 90.000,E1 119.077} C_DIS
LIN {X -0.005,Y -703.782,Z 1245.456,A 0.000,B 0.000,C 90.000,E1 118.153} C_DIS
LIN {X 0.184,Y -704.727,Z 1245.451,A 0.000,B 0.000,C 90.000,E1 117.206} C_DIS
LIN {X -0.209,Y -705.240,Z 1245.447,A 0.000,B 0.000,C 90.000,E1 116.539} C_DIS
LIN {X -0.285,Y -705.499,Z 1245.443,A 0.000,B 0.000,C 90.000,E1 115.848} C_DIS
LIN {X -0.354,Y -705.363,Z 1245.440,A 0.000,B 0.000,C 90.000,E1 115.155} C_DIS
LIN {X 0.224,Y -705.002,Z 1245.437,A 0.000,B 0.000,C 90.000,E1 114.643} C_DIS
LIN {X -0.134,Y -704.280,Z 1245.434,A 0.000,B 0.000,C 90.000,E1 114.207} C_DIS
LIN {X 0.150,Y -703.838,Z 1245.433,A 0.000,B 0.000,C 90.000,E1 113.951} C_DIS
LIN {X -0.075,Y -701.364,Z 1245.430,A 0.000,B 0.000,C 90.000,E1 113.387} C_DIS
LIN {X 0.063,Y -700.622,Z 1245.429,A 0.000,B 0.000,C 90.000,E1 113.259} C_DIS
LIN {X 0.102,Y -695.390,Z 1245.426,A 0.000,B 0.000,C 90.000,E1 112.717} C_DIS
LIN {X 0.231,Y -693.601,Z 1245.426,A 0.000,B 0.000,C 90.000,E1 112.589} C_DIS
LIN {X 0.127,Y -688.357,Z 1245.425,A 0.000,B 0.000,C 90.000,E1 112.408} C_DIS
LIN {X 0.329,Y -686.618,Z 1245.424,A 0.000,B 0.000,C 90.000,E1 112.333} C_DIS
LIN {X -0.018,Y -685.346,Z 1245.424,A 0.000,B 0.000,C 90.000,E1 112.333} C_DIS
LIN {X -0.072,Y -676.723,Z 1245.424,A 0.000,B 0.000,C 90.000,E1 112.259} C_DIS
LIN {X -0.114,Y -624.252,Z 1245.424,A 0.000,B 0.000,C 90.000,E1 112.259} C_DIS
LIN {X 0.005,Y -620.970,Z 1245.422,A 0.000,B 0.000,C 90.000,E1 112.025} C_DIS
LIN {X -0.030,Y -620.922,Z 1245.422,A 0.000,B 0.000,C 90.000,E1 112.025} C_DIS
LIN {X -0.084,Y -619.922,Z 1245.421,A 0.000,B 0.000,C 90.000,E1 111.844} C_DIS
LIN {X -0.127,Y -619.912,Z 1245.421,A 0.000,B 0.000,C 90.000,E1 111.844} C_DIS
LIN {X 0.206,Y -620.301,Z 1245.420,A 0.000,B 0.000,C 90.000,E1 111.589} C_DIS
LIN {X -0.185,Y -621.412,Z 1245.419,A 0.000,B 0.000,C 90.000,E1 111.354} C_DIS
LIN {X -0.083,Y -628.227,Z 1245.411,A 0.000,B 0.000,C 90.000,E1 110.066} C_DIS
LIN {X -0.241,Y -630.808,Z 1245.409,A 0.000,B 0.000,C 90.000,E1 109.577} C_DIS
LIN {X 0.172,Y -634.356,Z 1245.404,A 0.000,B 0.000,C 90.000,E1 108.779} C_DIS
LIN {X -0.230,Y -643.704,Z 1245.393,A 0.000,B 0.000,C 90.000,E1 106.804} C_DIS
LIN {X 0.117,Y -647.107,Z 1245.389,A 0.000,B 0.000,C 90.000,E1 106.024} C_DIS
LIN {X -0.167,Y -649.223,Z 1245.386,A 0.000,B 0.000,C 90.000,E1 105.552} C_DIS
LIN {X 0.232,Y -651.943,Z 1245.382,A 0.000,B 0.000,C 90.000,E1 104.773} C_DIS
LIN {X -0.021,Y -653.452,Z 1245.380,A 0.000,B 0.000,C 90.000,E1 104.300} C_DIS
LIN {X 0.255,Y -655.271,Z 1245.375,A 0.000,B 0.000,C 90.000,E1 103.536} C_DIS
LIN {X 0.026,Y -656.154,Z 1245.373,A 0.000,B 0.000,C 90.000,E1 103.063} C_DIS
LIN {X -0.200,Y -656.730,Z 1245.370,A 0.000,B 0.000,C 90.000,E1 102.591} C_DIS
LIN {X -0.311,Y -656.930,Z 1245.369,A 0.000,B 0.000,C 90.000,E1 102.355} C_DIS
LIN {X 0.107,Y -657.037,Z 1245.366,A 0.000,B 0.000,C 90.000,E1 101.827} C_DIS
LIN {X -0.247,Y -656.774,Z 1245.363,A 0.000,B 0.000,C 90.000,E1 101.366} C_DIS
LIN {X 0.174,Y -656.196,Z 1245.360,A 0.000,B 0.000,C 90.000,E1 100.838} C_DIS
LIN {X -0.058,Y -655.343,Z 1245.358,A 0.000,B 0.000,C 90.000,E1 100.366} C_DIS
LIN {X -0.292,Y -654.866,Z 1245.356,A 0.000,B 0.000,C 90.000,E1 100.141} C_DIS
LIN {X 0.111,Y -653.590,Z 1245.354,A 0.000,B 0.000,C 90.000,E1 99.613} C_DIS
LIN {X -0.250,Y -651.874,Z 1245.351,A 0.000,B 0.000,C 90.000,E1 99.151} C_DIS
LIN {X 0.125,Y -649.782,Z 1245.348,A 0.000,B 0.000,C 90.000,E1 98.624} C_DIS
LIN {X -0.254,Y -647.377,Z 1245.345,A 0.000,B 0.000,C 90.000,E1 98.163} C_DIS
LIN {X 0.234,Y -646.106,Z 1245.344,A 0.000,B 0.000,C 90.000,E1 97.871} C_DIS
LIN {X -0.296,Y -642.326,Z 1245.340,A 0.000,B 0.000,C 90.000,E1 97.296} C_DIS
LIN {X -0.085,Y -638.909,Z 1245.338,A 0.000,B 0.000,C 90.000,E1 96.777} C_DIS
LIN {X 0.102,Y -635.181,Z 1245.335,A 0.000,B 0.000,C 90.000,E1 96.258} C_DIS
LIN {X 0.261,Y -630.847,Z 1245.332,A 0.000,B 0.000,C 90.000,E1 95.739} C_DIS
LIN {X 0.272,Y -624.781,Z 1245.329,A 0.000,B 0.000,C 90.000,E1 95.106} C_DIS
LIN {X -0.085,Y -618.121,Z 1245.325,A 0.000,B 0.000,C 90.000,E1 94.531} C_DIS
LIN {X -0.113,Y -611.045,Z 1245.322,A 0.000,B 0.000,C 90.000,E1 93.955} C_DIS
LIN {X 0.271,Y -603.663,Z 1245.319,A 0.000,B 0.000,C 90.000,E1 93.383} C_DIS
LIN {X -0.220,Y -595.940,Z 1245.316,A 0.000,B 0.000,C 90.000,E1 92.922} C_DIS
LIN {X 0.216,Y -587.835,Z 1245.314,A 0.000,B 0.000,C 90.000,E1 92.407} C_DIS
LIN {X -0.130,Y -582.772,Z 1245.312,A 0.000,B 0.000,C 90.000,E1 92.178} C_DIS
LIN {X -0.077,Y -570.257,Z 1245.309,A 0.000,B 0.000,C 90.000,E1 91.661} C_DIS
LIN {X 0.250,Y -567.869,Z 1245.308,A 0.000,B 0.000,C 90.000,E1 91.489} C_DIS
LIN {X 0.193,Y -567.778,Z 1245.308,A 0.000,B 0.000,C 90.000,E1 91.489} C_DIS
LIN {X 0.241,Y -567.526,Z 1245.308,A 0.000,B 0.000,C 90.000,E1 91.375} C_DIS
LIN {X 0.023,Y -566.473,Z 1245.306,A 0.000,B 0.000,C 90.000,E1 91.088} C_DIS
LIN {X 0.032,Y -566.506,Z 1245.303,A 0.000,B 0.000,C 90.000,E1 90.573} C_DIS
LIN {X 0.175,Y -567.680,Z 1245.294,A 0.000,B 0.000,C 90.000,E1 88.912} C_DIS
LIN {X -0.217,Y -568.883,Z 1245.285,A 0.000,B 0.000,C 90.000,E1 87.306} C_DIS
LIN {X -0.138,Y -571.082,Z 1245.271,A 0.000,B 0.000,C 90.000,E1 84.837} C_DIS
LIN {X 0.075,Y -572.451,Z 1245.264,A 0.000,B 0.000,C 90.000,E1 83.451} C_DIS
LIN {X 0.064,Y -574.417,Z 1245.253,A 0.000,B 0.000,C 90.000,E1 81.546} C_DIS
LIN {X -0.144,Y -575.720,Z 1245.246,A 0.000,B 0.000,C 90.000,E1 80.208} C_DIS
LIN {X 0.025,Y -576.527,Z 1245.240,A 0.000,B 0.000,C 90.000,E1 79.106} C_DIS
LIN {X -0.041,Y -577.514,Z 1245.232,A 0.000,B 0.000,C 90.000,E1 77.757} C_DIS
LIN {X -0.088,Y -578.438,Z 1245.224,A 0.000,B 0.000,C 90.000,E1 76.408} C_DIS
LIN {X 0.015,Y -579.329,Z 1245.217,A 0.000,B 0.000,C 90.000,E1 75.046} C_DIS
LIN {X -0.049,Y -580.205,Z 1245.208,A 0.000,B 0.000,C 90.000,E1 73.433} C_DIS
LIN {X 0.248,Y -580.952,Z 1245.200,A 0.000,B 0.000,C 90.000,E1 72.054} C_DIS
LIN {X -0.002,Y -581.848,Z 1245.193,A 0.000,B 0.000,C 90.000,E1 70.732} C_DIS
LIN {X 0.263,Y -583.311,Z 1245.180,A 0.000,B 0.000,C 90.000,E1 68.284} C_DIS
LIN {X -0.038,Y -584.698,Z 1245.169,A 0.000,B 0.000,C 90.000,E1 66.433} C_DIS
LIN {X -0.249,Y -586.091,Z 1245.160,A 0.000,B 0.000,C 90.000,E1 64.845} C_DIS
LIN {X 0.025,Y -588.253,Z 1245.147,A 0.000,B 0.000,C 90.000,E1 62.410} C_DIS
LIN {X 0.158,Y -589.898,Z 1245.138,A 0.000,B 0.000,C 90.000,E1 60.795} C_DIS
LIN {X 0.201,Y -591.293,Z 1245.130,A 0.000,B 0.000,C 90.000,E1 59.459} C_DIS
LIN {X 0.274,Y -592.653,Z 1245.123,A 0.000,B 0.000,C 90.000,E1 58.122} C_DIS
LIN {X -0.028,Y -593.720,Z 1245.117,A 0.000,B 0.000,C 90.000,E1 57.089} C_DIS
LIN {X -0.202,Y -595.132,Z 1245.108,A 0.000,B 0.000,C 90.000,E1 55.515} C_DIS
LIN {X -0.246,Y -596.254,Z 1245.101,A 0.000,B 0.000,C 90.000,E1 54.196} C_DIS
LIN {X 0.088,Y -596.898,Z 1245.097,A 0.000,B 0.000,C 90.000,E1 53.371} C_DIS
LIN {X -0.066,Y -597.966,Z 1245.089,A 0.000,B 0.000,C 90.000,E1 52.065} C_DIS
LIN {X -0.060,Y -598.796,Z 1245.083,A 0.000,B 0.000,C 90.000,E1 51.009} C_DIS
LIN {X -0.403,Y -599.643,Z 1245.075,A 0.000,B 0.000,C 90.000,E1 49.461} C_DIS
LIN {X 0.263,Y -600.179,Z 1245.067,A 0.000,B 0.000,C 90.000,E1 48.081} C_DIS
LIN {X 0.070,Y -600.508,Z 1245.063,A 0.000,B 0.000,C 90.000,E1 47.310} C_DIS
LIN {X -0.332,Y -600.681,Z 1245.057,A 0.000,B 0.000,C 90.000,E1 46.296} C_DIS
LIN {X -0.316,Y -600.801,Z 1245.051,A 0.000,B 0.000,C 90.000,E1 45.243} C_DIS
LIN {X -0.296,Y -600.714,Z 1245.045,A 0.000,B 0.000,C 90.000,E1 44.190} C_DIS
LIN {X 0.155,Y -600.494,Z 1245.040,A 0.000,B 0.000,C 90.000,E1 43.095} C_DIS
LIN {X -0.244,Y -600.120,Z 1245.034,A 0.000,B 0.000,C 90.000,E1 42.081} C_DIS
LIN {X -0.024,Y -599.535,Z 1245.026,A 0.000,B 0.000,C 90.000,E1 40.744} C_DIS
LIN {X -0.142,Y -598.863,Z 1245.019,A 0.000,B 0.000,C 90.000,E1 39.439} C_DIS
LIN {X -0.122,Y -597.998,Z 1245.013,A 0.000,B 0.000,C 90.000,E1 38.382} C_DIS
LIN {X -0.017,Y -597.088,Z 1245.007,A 0.000,B 0.000,C 90.000,E1 37.317} C_DIS
LIN {X 0.205,Y -596.224,Z 1245.003,A 0.000,B 0.000,C 90.000,E1 36.503} C_DIS
LIN {X -0.061,Y -594.724,Z 1244.997,A 0.000,B 0.000,C 90.000,E1 35.471} C_DIS
LIN {X 0.000,Y -592.943,Z 1244.991,A 0.000,B 0.000,C 90.000,E1 34.405} C_DIS
LIN {X -0.303,Y -590.884,Z 1244.985,A 0.000,B 0.000,C 90.000,E1 33.372} C_DIS
LIN {X -0.017,Y -588.929,Z 1244.981,A 0.000,B 0.000,C 90.000,E1 32.546} C_DIS
LIN {X -0.067,Y -586.682,Z 1244.976,A 0.000,B 0.000,C 90.000,E1 31.750} C_DIS
LIN {X 0.167,Y -584.127,Z 1244.972,A 0.000,B 0.000,C 90.000,E1 30.924} C_DIS
LIN {X -0.091,Y -582.194,Z 1244.969,A 0.000,B 0.000,C 90.000,E1 30.413} C_DIS
LIN {X 0.084,Y -579.016,Z 1244.964,A 0.000,B 0.000,C 90.000,E1 29.589} C_DIS
LIN {X -0.350,Y -575.226,Z 1244.960,A 0.000,B 0.000,C 90.000,E1 28.821} C_DIS
LIN {X -0.124,Y -570.400,Z 1244.955,A 0.000,B 0.000,C 90.000,E1 27.847} C_DIS
LIN {X 0.218,Y -566.446,Z 1244.951,A 0.000,B 0.000,C 90.000,E1 27.129} C_DIS
LIN {X -0.239,Y -562.199,Z 1244.947,A 0.000,B 0.000,C 90.000,E1 26.488} C_DIS
LIN {X -0.124,Y -558.590,Z 1244.944,A 0.000,B 0.000,C 90.000,E1 25.924} C_DIS
LIN {X 0.314,Y -555.739,Z 1244.942,A 0.000,B 0.000,C 90.000,E1 25.463} C_DIS
LIN {X -0.120,Y -551.674,Z 1244.939,A 0.000,B 0.000,C 90.000,E1 24.951} C_DIS
LIN {X -0.201,Y -546.215,Z 1244.935,A 0.000,B 0.000,C 90.000,E1 24.259} C_DIS
LIN {X -0.071,Y -542.749,Z 1244.932,A 0.000,B 0.000,C 90.000,E1 23.823} C_DIS
LIN {X -0.024,Y -536.767,Z 1244.929,A 0.000,B 0.000,C 90.000,E1 23.131} C_DIS
LIN {X -0.268,Y -530.600,Z 1244.925,A 0.000,B 0.000,C 90.000,E1 22.461} C_DIS
LIN {X -0.083,Y -521.228,Z 1244.919,A 0.000,B 0.000,C 90.000,E1 21.461} C_DIS
LIN {X 0.111,Y -513.139,Z 1244.915,A 0.000,B 0.000,C 90.000,E1 20.610} C_DIS
LIN {X 0.063,Y -507.618,Z 1244.912,A 0.000,B 0.000,C 90.000,E1 20.066} C_DIS
LIN {X 0.094,Y -498.115,Z 1244.906,A 0.000,B 0.000,C 90.000,E1 19.141} C_DIS
LIN {X -0.150,Y -488.173,Z 1244.901,A 0.000,B 0.000,C 90.000,E1 18.236} C_DIS
LIN {X -0.198,Y -480.837,Z 1244.898,A 0.000,B 0.000,C 90.000,E1 17.583} C_DIS
LIN {X -0.060,Y -464.583,Z 1244.890,A 0.000,B 0.000,C 90.000,E1 16.134} C_DIS
LIN {X -0.041,Y -448.266,Z 1244.881,A 0.000,B 0.000,C 90.000,E1 14.647} C_DIS
LIN {X -0.143,Y -429.337,Z 1244.871,A 0.000,B 0.000,C 90.000,E1 12.827} C_DIS
LIN {X 0.058,Y -409.335,Z 1244.859,A 0.000,B 0.000,C 90.000,E1 10.658} C_DIS
LIN {X 0.214,Y -400.839,Z 1244.854,A 0.000,B 0.000,C 90.000,E1 9.670} C_DIS
LIN {X -0.140,Y -397.089,Z 1244.851,A 0.000,B 0.000,C 90.000,E1 9.208} C_DIS
LIN {X -0.119,Y -396.022,Z 1244.850,A 0.000,B 0.000,C 90.000,E1 9.029} C_DIS
LIN {X -0.068,Y -394.399,Z 1244.848,A 0.000,B 0.000,C 90.000,E1 8.681} C_DIS
LIN {X -0.106,Y -394.388,Z 1244.848,A 0.000,B 0.000,C 90.000,E1 8.681} C_DIS
LIN {X 0.028,Y -394.278,Z 1244.848,A 0.000,B 0.000,C 90.000,E1 8.568} C_DIS
LIN {X -0.009,Y -394.294,Z 1244.848,A 0.000,B 0.000,C 90.000,E1 8.568} C_DIS
LIN {X -0.139,Y -396.482,Z 1244.845,A 0.000,B 0.000,C 90.000,E1 8.106} C_DIS
LIN {X -0.149,Y -400.973,Z 1244.842,A 0.000,B 0.000,C 90.000,E1 7.644} C_DIS
LIN {X -0.096,Y -406.365,Z 1244.840,A 0.000,B 0.000,C 90.000,E1 7.239} C_DIS
LIN {X 0.134,Y -412.700,Z 1244.838,A 0.000,B 0.000,C 90.000,E1 6.777} C_DIS
LIN {X 0.072,Y -424.076,Z 1244.833,A 0.000,B 0.000,C 90.000,E1 5.967} C_DIS
LIN {X -0.064,Y -430.434,Z 1244.831,A 0.000,B 0.000,C 90.000,E1 5.511} C_DIS
LIN {X 0.035,Y -439.772,Z 1244.827,A 0.000,B 0.000,C 90.000,E1 4.759} C_DIS
LIN {X 0.060,Y -449.200,Z 1244.822,A 0.000,B 0.000,C 90.000,E1 4.012} C_DIS
LIN {X -0.128,Y -461.468,Z 1244.817,A 0.000,B 0.000,C 90.000,E1 3.037} C_DIS
LIN {X -0.035,Y -467.484,Z 1244.814,A 0.000,B 0.000,C 90.000,E1 2.522} C_DIS
LIN {X -0.055,Y -473.303,Z 1244.811,A 0.000,B 0.000,C 90.000,E1 2.007} C_DIS
LIN {X -0.005,Y -478.754,Z 1244.808,A 0.000,B 0.000,C 90.000,E1 1.489} C_DIS
LIN {X -0.002,Y -485.361,Z 1244.804,A 0.000,B 0.000,C 90.000,E1 0.802} C_DIS
LIN {X 0.000,Y -492.444,Z 1244.800,A 0.000,B 0.000,C 90.000,E1 360.000} C_DIS
LIN {X 0.039,Y -496.767,Z 1244.797,A 0.000,B 0.000,C 90.000,E1 359.484} C_DIS
LIN {X -0.208,Y -503.459,Z 1244.792,A 0.000,B 0.000,C 90.000,E1 358.625} C_DIS
LIN {X 0.088,Y -507.750,Z 1244.789,A 0.000,B 0.000,C 90.000,E1 357.993} C_DIS
LIN {X 0.103,Y -512.662,Z 1244.785,A 0.000,B 0.000,C 90.000,E1 357.249} C_DIS
LIN {X 0.185,Y -517.340,Z 1244.781,A 0.000,B 0.000,C 90.000,E1 356.502} C_DIS
LIN {X 0.087,Y -520.832,Z 1244.777,A 0.000,B 0.000,C 90.000,E1 355.927} C_DIS
LIN {X 0.209,Y -524.803,Z 1244.773,A 0.000,B 0.000,C 90.000,E1 355.184} C_DIS
LIN {X -0.072,Y -528.431,Z 1244.769,A 0.000,B 0.000,C 90.000,E1 354.489} C_DIS
LIN {X -0.089,Y -531.155,Z 1244.766,A 0.000,B 0.000,C 90.000,E1 353.913} C_DIS
LIN {X -0.086,Y -533.710,Z 1244.763,A 0.000,B 0.000,C 90.000,E1 353.337} C_DIS
LIN {X -0.069,Y -536.080,Z 1244.760,A 0.000,B 0.000,C 90.000,E1 352.761} C_DIS
LIN {X 0.020,Y -539.295,Z 1244.755,A 0.000,B 0.000,C 90.000,E1 351.894} C_DIS
LIN {X 0.217,Y -543.154,Z 1244.749,A 0.000,B 0.000,C 90.000,E1 350.735} C_DIS
LIN {X -0.162,Y -545.738,Z 1244.744,A 0.000,B 0.000,C 90.000,E1 349.926} C_DIS
LIN {X 0.219,Y -548.896,Z 1244.738,A 0.000,B 0.000,C 90.000,E1 348.757} C_DIS
LIN {X 0.111,Y -551.732,Z 1244.731,A 0.000,B 0.000,C 90.000,E1 347.645} C_DIS
LIN {X 0.290,Y -554.819,Z 1244.724,A 0.000,B 0.000,C 90.000,E1 346.228} C_DIS
LIN {X -0.283,Y -557.037,Z 1244.718,A 0.000,B 0.000,C 90.000,E1 345.172} C_DIS
LIN {X 0.134,Y -559.442,Z 1244.710,A 0.000,B 0.000,C 90.000,E1 343.740} C_DIS
LIN {X 0.161,Y -560.650,Z 1244.705,A 0.000,B 0.000,C 90.000,E1 342.906} C_DIS
LIN {X -0.032,Y -562.078,Z 1244.699,A 0.000,B 0.000,C 90.000,E1 341.819} C_DIS
LIN {X -0.204,Y -563.157,Z 1244.693,A 0.000,B 0.000,C 90.000,E1 340.732} C_DIS
LIN {X 0.035,Y -563.701,Z 1244.688,A 0.000,B 0.000,C 90.000,E1 339.880} C_DIS
LIN {X -0.249,Y -563.991,Z 1244.684,A 0.000,B 0.000,C 90.000,E1 339.082} C_DIS
LIN {X -0.123,Y -564.049,Z 1244.681,A 0.000,B 0.000,C 90.000,E1 338.518} C_DIS
LIN {X 0.121,Y -563.776,Z 1244.676,A 0.000,B 0.000,C 90.000,E1 337.667} C_DIS
LIN {X 0.249,Y -563.441,Z 1244.673,A 0.000,B 0.000,C 90.000,E1 337.102} C_DIS
LIN {X -0.240,Y -562.262,Z 1244.667,A 0.000,B 0.000,C 90.000,E1 336.049} C_DIS
LIN {X -0.121,Y -561.518,Z 1244.664,A 0.000,B 0.000,C 90.000,E1 335.485} C_DIS
LIN {X -0.209,Y -560.040,Z 1244.659,A 0.000,B 0.000,C 90.000,E1 334.665} C_DIS
LIN {X 0.226,Y -557.635,Z 1244.653,A 0.000,B 0.000,C 90.000,E1 333.512} C_DIS
LIN {X 0.018,Y -557.016,Z 1244.651,A 0.000,B 0.000,C 90.000,E1 333.256} C_DIS
LIN {X 0.132,Y -554.518,Z 1244.647,A 0.000,B 0.000,C 90.000,E1 332.410} C_DIS
LIN {X -0.040,Y -551.751,Z 1244.642,A 0.000,B 0.000,C 90.000,E1 331.591} C_DIS
LIN {X 0.280,Y -548.292,Z 1244.638,A 0.000,B 0.000,C 90.000,E1 330.717} C_DIS
LIN {X -0.056,Y -544.926,Z 1244.634,A 0.000,B 0.000,C 90.000,E1 330.049} C_DIS
LIN {X 0.050,Y -541.054,Z 1244.630,A 0.000,B 0.000,C 90.000,E1 329.331} C_DIS
LIN {X 0.253,Y -535.658,Z 1244.625,A 0.000,B 0.000,C 90.000,E1 328.456} C_DIS
LIN {X -0.339,Y -529.921,Z 1244.620,A 0.000,B 0.000,C 90.000,E1 327.661} C_DIS
LIN {X 0.025,Y -523.745,Z 1244.615,A 0.000,B 0.000,C 90.000,E1 326.755} C_DIS
LIN {X 0.030,Y -517.503,Z 1244.610,A 0.000,B 0.000,C 90.000,E1 325.881} C_DIS
LIN {X -0.096,Y -513.723,Z 1244.607,A 0.000,B 0.000,C 90.000,E1 325.308} C_DIS
LIN {X -0.055,Y -510.690,Z 1244.604,A 0.000,B 0.000,C 90.000,E1 324.769} C_DIS
LIN {X 0.191,Y -508.125,Z 1244.601,A 0.000,B 0.000,C 90.000,E1 324.116} C_DIS
LIN {X -0.194,Y -506.291,Z 1244.597,A 0.000,B 0.000,C 90.000,E1 323.417} C_DIS
LIN {X 0.010,Y -505.280,Z 1244.593,A 0.000,B 0.000,C 90.000,E1 322.798} C_DIS
LIN {X 0.108,Y -504.700,Z 1244.590,A 0.000,B 0.000,C 90.000,E1 322.190} C_DIS
LIN {X -0.214,Y -504.400,Z 1244.585,A 0.000,B 0.000,C 90.000,E1 321.331} C_DIS
LIN {X 0.089,Y -505.253,Z 1244.570,A 0.000,B 0.000,C 90.000,E1 318.609} C_DIS
LIN {X -0.180,Y -505.716,Z 1244.562,A 0.000,B 0.000,C 90.000,E1 317.148} C_DIS
LIN {X -0.098,Y -506.195,Z 1244.554,A 0.000,B 0.000,C 90.000,E1 315.648} C_DIS
LIN {X -0.141,Y -506.627,Z 1244.544,A 0.000,B 0.000,C 90.000,E1 313.866} C_DIS
LIN {X -0.157,Y -507.194,Z 1244.534,A 0.000,B 0.000,C 90.000,E1 312.081} C_DIS
LIN {X 0.325,Y -507.695,Z 1244.526,A 0.000,B 0.000,C 90.000,E1 310.539} C_DIS
LIN {X -0.140,Y -507.993,Z 1244.519,A 0.000,B 0.000,C 90.000,E1 309.402} C_DIS
LIN {X -0.093,Y -508.553,Z 1244.507,A 0.000,B 0.000,C 90.000,E1 307.317} C_DIS
LIN {X 0.249,Y -508.864,Z 1244.501,A 0.000,B 0.000,C 90.000,E1 306.091} C_DIS
LIN {X 0.201,Y -509.110,Z 1244.492,A 0.000,B 0.000,C 90.000,E1 304.612} C_DIS
LIN {X -0.130,Y -509.331,Z 1244.484,A 0.000,B 0.000,C 90.000,E1 303.166} C_DIS
LIN {X -0.032,Y -509.474,Z 1244.476,A 0.000,B 0.000,C 90.000,E1 301.671} C_DIS
LIN {X 0.026,Y -509.472,Z 1244.464,A 0.000,B 0.000,C 90.000,E1 299.589} C_DIS
LIN {X -0.037,Y -509.410,Z 1244.458,A 0.000,B 0.000,C 90.000,E1 298.409} C_DIS
LIN {X -0.014,Y -509.317,Z 1244.450,A 0.000,B 0.000,C 90.000,E1 296.924} C_DIS
LIN {X -0.063,Y -509.396,Z 1244.435,A 0.000,B 0.000,C 90.000,E1 294.259} C_DIS
LIN {X -0.218,Y -509.403,Z 1244.430,A 0.000,B 0.000,C 90.000,E1 293.387} C_DIS
LIN {X 0.205,Y -509.203,Z 1244.423,A 0.000,B 0.000,C 90.000,E1 292.153} C_DIS
LIN {X 0.048,Y -508.826,Z 1244.418,A 0.000,B 0.000,C 90.000,E1 291.280} C_DIS
LIN {X -0.196,Y -508.304,Z 1244.412,A 0.000,B 0.000,C 90.000,E1 290.120} C_DIS
LIN {X 0.062,Y -507.536,Z 1244.402,A 0.000,B 0.000,C 90.000,E1 288.308} C_DIS
LIN {X 0.215,Y -506.977,Z 1244.394,A 0.000,B 0.000,C 90.000,E1 286.804} C_DIS
LIN {X -0.221,Y -506.533,Z 1244.387,A 0.000,B 0.000,C 90.000,E1 285.662} C_DIS
LIN {X 0.248,Y -505.728,Z 1244.379,A 0.000,B 0.000,C 90.000,E1 284.120} C_DIS
LIN {X 0.028,Y -504.543,Z 1244.369,A 0.000,B 0.000,C 90.000,E1 282.355} C_DIS
LIN {X 0.046,Y -502.754,Z 1244.355,A 0.000,B 0.000,C 90.000,E1 279.962} C_DIS
LIN {X 0.131,Y -501.685,Z 1244.347,A 0.000,B 0.000,C 90.000,E1 278.454} C_DIS
LIN {X -0.160,Y -500.309,Z 1244.334,A 0.000,B 0.000,C 90.000,E1 276.087} C_DIS
LIN {X -0.188,Y -499.519,Z 1244.325,A 0.000,B 0.000,C 90.000,E1 274.588} C_DIS
LIN {X -0.045,Y -498.297,Z 1244.314,A 0.000,B 0.000,C 90.000,E1 272.465} C_DIS
LIN {X 0.176,Y -496.832,Z 1244.304,A 0.000,B 0.000,C 90.000,E1 270.630} C_DIS
LIN {X -0.002,Y -495.830,Z 1244.295,A 0.000,B 0.000,C 90.000,E1 269.141} C_DIS
LIN {X 0.163,Y -494.637,Z 1244.285,A 0.000,B 0.000,C 90.000,E1 267.306} C_DIS
LIN {X -0.101,Y -494.305,Z 1244.282,A 0.000,B 0.000,C 90.000,E1 266.731} C_DIS
LIN {X 0.058,Y -493.311,Z 1244.272,A 0.000,B 0.000,C 90.000,E1 264.894} C_DIS
LIN {X -0.097,Y -492.344,Z 1244.263,A 0.000,B 0.000,C 90.000,E1 263.394} C_DIS
LIN {X -0.162,Y -491.391,Z 1244.257,A 0.000,B 0.000,C 90.000,E1 262.186} C_DIS
LIN {X 0.080,Y -489.627,Z 1244.246,A 0.000,B 0.000,C 90.000,E1 260.330} C_DIS
LIN {X -0.119,Y -486.851,Z 1244.228,A 0.000,B 0.000,C 90.000,E1 256.992} C_DIS
LIN {X 0.062,Y -485.321,Z 1244.214,A 0.000,B 0.000,C 90.000,E1 254.519} C_DIS
LIN {X -0.208,Y -484.616,Z 1244.207,A 0.000,B 0.000,C 90.000,E1 253.323} C_DIS
LIN {X -0.020,Y -483.417,Z 1244.195,A 0.000,B 0.000,C 90.000,E1 251.148} C_DIS
LIN {X -0.159,Y -482.635,Z 1244.187,A 0.000,B 0.000,C 90.000,E1 249.625} C_DIS
LIN {X 0.126,Y -481.689,Z 1244.177,A 0.000,B 0.000,C 90.000,E1 247.741} C_DIS
LIN {X -0.140,Y -480.750,Z 1244.168,A 0.000,B 0.000,C 90.000,E1 246.230} C_DIS
LIN {X 0.020,Y -479.644,Z 1244.159,A 0.000,B 0.000,C 90.000,E1 244.665} C_DIS
LIN {X -0.072,Y -478.542,Z 1244.151,A 0.000,B 0.000,C 90.000,E1 243.127} C_DIS
LIN {X 0.038,Y -477.361,Z 1244.142,A 0.000,B 0.000,C 90.000,E1 241.563} C_DIS
LIN {X 0.126,Y -476.047,Z 1244.133,A 0.000,B 0.000,C 90.000,E1 239.999} C_DIS
LIN {X 0.013,Y -474.554,Z 1244.125,A 0.000,B 0.000,C 90.000,E1 238.456} C_DIS
LIN {X -0.130,Y -473.176,Z 1244.116,A 0.000,B 0.000,C 90.000,E1 236.914} C_DIS
LIN {X -0.059,Y -471.010,Z 1244.102,A 0.000,B 0.000,C 90.000,E1 234.402} C_DIS
LIN {X -0.156,Y -469.223,Z 1244.088,A 0.000,B 0.000,C 90.000,E1 231.904} C_DIS
LIN {X 0.070,Y -467.797,Z 1244.078,A 0.000,B 0.000,C 90.000,E1 229.989} C_DIS
LIN {X 0.143,Y -466.655,Z 1244.069,A 0.000,B 0.000,C 90.000,E1 228.405} C_DIS
LIN {X -0.093,Y -465.309,Z 1244.059,A 0.000,B 0.000,C 90.000,E1 226.539} C_DIS
LIN {X 0.057,Y -463.390,Z 1244.036,A 0.000,B 0.000,C 90.000,E1 222.405} C_DIS
LIN {X -0.163,Y -464.551,Z 1244.000,A 0.000,B 0.000,C 90.000,E1 216.091} C_DIS
LIN {X 0.035,Y -467.406,Z 1243.978,A 0.000,B 0.000,C 90.000,E1 211.957} C_DIS
LIN {X 0.097,Y -469.638,Z 1243.965,A 0.000,B 0.000,C 90.000,E1 209.745} C_DIS
LIN {X -0.081,Y -472.671,Z 1243.951,A 0.000,B 0.000,C 90.000,E1 207.257} C_DIS
LIN {X 0.135,Y -474.587,Z 1243.943,A 0.000,B 0.000,C 90.000,E1 205.668} C_DIS
LIN {X -0.139,Y -479.043,Z 1243.925,A 0.000,B 0.000,C 90.000,E1 202.589} C_DIS
LIN {X 0.281,Y -484.985,Z 1243.907,A 0.000,B 0.000,C 90.000,E1 199.141} C_DIS
LIN {X -0.184,Y -491.492,Z 1243.890,A 0.000,B 0.000,C 90.000,E1 196.134} C_DIS
LIN {X -0.090,Y -495.678,Z 1243.879,A 0.000,B 0.000,C 90.000,E1 194.300} C_DIS
LIN {X -0.010,Y -499.919,Z 1243.869,A 0.000,B 0.000,C 90.000,E1 192.479} C_DIS
LIN {X 0.164,Y -504.349,Z 1243.859,A 0.000,B 0.000,C 90.000,E1 190.658} C_DIS
LIN {X 0.249,Y -508.934,Z 1243.849,A 0.000,B 0.000,C 90.000,E1 188.859} C_DIS
LIN {X -0.037,Y -512.807,Z 1243.841,A 0.000,B 0.000,C 90.000,E1 187.409} C_DIS
LIN {X 0.215,Y -515.880,Z 1243.835,A 0.000,B 0.000,C 90.000,E1 186.201} C_DIS
LIN {X -0.021,Y -519.639,Z 1243.826,A 0.000,B 0.000,C 90.000,E1 184.759} C_DIS
LIN {X 0.248,Y -523.452,Z 1243.818,A 0.000,B 0.000,C 90.000,E1 183.269} C_DIS
LIN {X 0.062,Y -527.891,Z 1243.809,A 0.000,B 0.000,C 90.000,E1 181.547} C_DIS
LIN {X -0.064,Y -532.235,Z 1243.799,A 0.000,B 0.000,C 90.000,E1 179.828} C_DIS
LIN {X -0.097,Y -535.050,Z 1243.793,A 0.000,B 0.000,C 90.000,E1 178.682} C_DIS
LIN {X -0.079,Y -537.131,Z 1243.788,A 0.000,B 0.000,C 90.000,E1 177.822} C_DIS
LIN {X -0.010,Y -540.402,Z 1243.780,A 0.000,B 0.000,C 90.000,E1 176.388} C_DIS
LIN {X 0.169,Y -544.059,Z 1243.771,A 0.000,B 0.000,C 90.000,E1 174.666} C_DIS
LIN {X -0.179,Y -546.381,Z 1243.764,A 0.000,B 0.000,C 90.000,E1 173.571} C_DIS
LIN {X 0.020,Y -548.088,Z 1243.760,A 0.000,B 0.000,C 90.000,E1 172.704} C_DIS
LIN {X -0.202,Y -550.273,Z 1243.753,A 0.000,B 0.000,C 90.000,E1 171.602} C_DIS
LIN {X -0.248,Y -553.324,Z 1243.744,A 0.000,B 0.000,C 90.000,E1 169.926} C_DIS
LIN {X -0.172,Y -555.776,Z 1243.736,A 0.000,B 0.000,C 90.000,E1 168.522} C_DIS
LIN {X 0.090,Y -558.613,Z 1243.727,A 0.000,B 0.000,C 90.000,E1 166.825} C_DIS
LIN {X 0.285,Y -561.981,Z 1243.716,A 0.000,B 0.000,C 90.000,E1 164.866} C_DIS
LIN {X -0.034,Y -566.961,Z 1243.702,A 0.000,B 0.000,C 90.000,E1 162.417} C_DIS
LIN {X -0.166,Y -571.371,Z 1243.693,A 0.000,B 0.000,C 90.000,E1 160.786} C_DIS
LIN {X 0.159,Y -576.026,Z 1243.686,A 0.000,B 0.000,C 90.000,E1 159.390} C_DIS
LIN {X -0.127,Y -582.582,Z 1243.677,A 0.000,B 0.000,C 90.000,E1 157.794} C_DIS
LIN {X -0.210,Y -591.831,Z 1243.665,A 0.000,B 0.000,C 90.000,E1 155.793} C_DIS
LIN {X 0.317,Y -599.429,Z 1243.657,A 0.000,B 0.000,C 90.000,E1 154.152} C_DIS
LIN {X 0.067,Y -603.830,Z 1243.651,A 0.000,B 0.000,C 90.000,E1 153.256} C_DIS
LIN {X -0.210,Y -609.808,Z 1243.644,A 0.000,B 0.000,C 90.000,E1 151.975} C_DIS
LIN {X -0.080,Y -614.365,Z 1243.638,A 0.000,B 0.000,C 90.000,E1 150.923} C_DIS
LIN {X 0.097,Y -619.928,Z 1243.631,A 0.000,B 0.000,C 90.000,E1 149.616} C_DIS
LIN {X -0.162,Y -623.255,Z 1243.627,A 0.000,B 0.000,C 90.000,E1 148.869} C_DIS
LIN {X 0.302,Y -630.585,Z 1243.617,A 0.000,B 0.000,C 90.000,E1 147.041} C_DIS
LIN {X -0.360,Y -634.495,Z 1243.611,A 0.000,B 0.000,C 90.000,E1 146.087} C_DIS
LIN {X -0.096,Y -638.193,Z 1243.606,A 0.000,B 0.000,C 90.000,E1 145.055} C_DIS
LIN {X 0.188,Y -640.793,Z 1243.602,A 0.000,B 0.000,C 90.000,E1 144.276} C_DIS
LIN {X -0.017,Y -643.245,Z 1243.598,A 0.000,B 0.000,C 90.000,E1 143.543} C_DIS
LIN {X 0.261,Y -646.943,Z 1243.591,A 0.000,B 0.000,C 90.000,E1 142.271} C_DIS
LIN {X 0.048,Y -649.718,Z 1243.585,A 0.000,B 0.000,C 90.000,E1 141.295} C_DIS
LIN {X 0.383,Y -652.293,Z 1243.580,A 0.000,B 0.000,C 90.000,E1 140.275} C_DIS
LIN {X -0.274,Y -656.034,Z 1243.571,A 0.000,B 0.000,C 90.000,E1 138.852} C_DIS
LIN {X 0.041,Y -659.026,Z 1243.564,A 0.000,B 0.000,C 90.000,E1 137.595} C_DIS
LIN {X -0.041,Y -661.926,Z 1243.558,A 0.000,B 0.000,C 90.000,E1 136.377} C_DIS
LIN {X -0.118,Y -667.445,Z 1243.546,A 0.000,B 0.000,C 90.000,E1 134.190} C_DIS
LIN {X -0.098,Y -670.641,Z 1243.539,A 0.000,B 0.000,C 90.000,E1 132.975} C_DIS
LIN {X 0.025,Y -674.492,Z 1243.531,A 0.000,B 0.000,C 90.000,E1 131.515} C_DIS
LIN {X -0.192,Y -678.939,Z 1243.521,A 0.000,B 0.000,C 90.000,E1 129.850} C_DIS
LIN {X -0.216,Y -683.239,Z 1243.512,A 0.000,B 0.000,C 90.000,E1 128.177} C_DIS
LIN {X -0.175,Y -686.922,Z 1243.504,A 0.000,B 0.000,C 90.000,E1 126.744} C_DIS
LIN {X -0.294,Y -689.201,Z 1243.499,A 0.000,B 0.000,C 90.000,E1 125.804} C_DIS
LIN {X 0.413,Y -692.388,Z 1243.491,A 0.000,B 0.000,C 90.000,E1 124.326} C_DIS
LIN {X 0.179,Y -694.958,Z 1243.484,A 0.000,B 0.000,C 90.000,E1 123.166} C_DIS
LIN {X 0.332,Y -696.883,Z 1243.479,A 0.000,B 0.000,C 90.000,E1 122.212} C_DIS
LIN {X -0.179,Y -699.547,Z 1243.471,A 0.000,B 0.000,C 90.000,E1 120.846} C_DIS
LIN {X 0.270,Y -701.275,Z 1243.466,A 0.000,B 0.000,C 90.000,E1 119.873} C_DIS
LIN {X -0.197,Y -703.122,Z 1243.460,A 0.000,B 0.000,C 90.000,E1 118.743} C_DIS
LIN {X 0.307,Y -704.270,Z 1243.454,A 0.000,B 0.000,C 90.000,E1 117.769} C_DIS
LIN {X -0.122,Y -705.152,Z 1243.449,A 0.000,B 0.000,C 90.000,E1 116.873} C_DIS
LIN {X 0.114,Y -705.515,Z 1243.445,A 0.000,B 0.000,C 90.000,E1 116.155} C_DIS
LIN {X -0.249,Y -705.629,Z 1243.443,A 0.000,B 0.000,C 90.000,E1 115.720} C_DIS
LIN {X -0.317,Y -705.378,Z 1243.439,A 0.000,B 0.000,C 90.000,E1 115.027} C_DIS
LIN {X 0.261,Y -704.984,Z 1243.436,A 0.000,B 0.000,C 90.000,E1 114.515} C_DIS
LIN {X -0.099,Y -704.193,Z 1243.434,A 0.000,B 0.000,C 90.000,E1 114.079} C_DIS
LIN {X 0.185,Y -703.483,Z 1243.432,A 0.000,B 0.000,C 90.000,E1 113.823} C_DIS
LIN {X -0.180,Y -701.490,Z 1243.430,A 0.000,B 0.000,C 90.000,E1 113.387} C_DIS
LIN {X -0.043,Y -700.737,Z 1243.429,A 0.000,B 0.000,C 90.000,E1 113.259} C_DIS
LIN {X 0.001,Y -695.356,Z 1243.426,A 0.000,B 0.000,C 90.000,E1 112.717} C_DIS
LIN {X 0.133,Y -693.520,Z 1243.426,A 0.000,B 0.000,C 90.000,E1 112.589} C_DIS
LIN {X 0.153,Y -688.503,Z 1243.425,A 0.000,B 0.000,C 90.000,E1 112.408} C_DIS
LIN {X 0.051,Y -685.769,Z 1243.424,A 0.000,B 0.000,C 90.000,E1 112.333} C_DIS
LIN {X 0.224,Y -681.998,Z 1243.424,A 0.000,B 0.000,C 90.000,E1 112.280} C_DIS
LIN {X -0.273,Y -677.289,Z 1243.424,A 0.000,B 0.000,C 90.000,E1 112.280} C_DIS
LIN {X -0.077,Y -623.228,Z 1243.424,A 0.000,B 0.000,C 90.000,E1 112.259} C_DIS
LIN {X 0.146,Y -620.104,Z 1243.422,A 0.000,B 0.000,C 90.000,E1 112.025} C_DIS
LIN {X 0.043,Y -618.806,Z 1243.421,A 0.000,B 0.000,C 90.000,E1 111.844} C_DIS
LIN {X -0.007,Y -618.803,Z 1243.421,A 0.000,B 0.000,C 90.000,E1 111.844} C_DIS
LIN {X 0.150,Y -618.793,Z 1243.421,A 0.000,B 0.000,C 90.000,E1 111.663} C_DIS
LIN {X 0.249,Y -619.448,Z 1243.419,A 0.000,B 0.000,C 90.000,E1 111.461} C_DIS
LIN {X -0.008,Y -621.152,Z 1243.417,A 0.000,B 0.000,C 90.000,E1 111.099} C_DIS
LIN {X 0.091,Y -625.986,Z 1243.412,A 0.000,B 0.000,C 90.000,E1 110.194} C_DIS
LIN {X -0.097,Y -628.543,Z 1243.409,A 0.000,B 0.000,C 90.000,E1 109.704} C_DIS
LIN {X 0.295,Y -632.085,Z 1243.405,A 0.000,B 0.000,C 90.000,E1 108.906} C_DIS
LIN {X -0.082,Y -635.483,Z 1243.401,A 0.000,B 0.000,C 90.000,E1 108.181} C_DIS
LIN {X -0.253,Y -637.707,Z 1243.398,A 0.000,B 0.000,C 90.000,E1 107.692} C_DIS
LIN {X -0.135,Y -642.498,Z 1243.393,A 0.000,B 0.000,C 90.000,E1 106.677} C_DIS
LIN {X 0.169,Y -644.775,Z 1243.390,A 0.000,B 0.000,C 90.000,E1 106.150} C_DIS
LIN {X 0.047,Y -646.916,Z 1243.387,A 0.000,B 0.000,C 90.000,E1 105.662} C_DIS
LIN {X 0.251,Y -649.758,Z 1243.383,A 0.000,B 0.000,C 90.000,E1 104.898} C_DIS
LIN {X 0.019,Y -651.975,Z 1243.379,A 0.000,B 0.000,C 90.000,E1 104.175} C_DIS
LIN {X -0.234,Y -653.217,Z 1243.376,A 0.000,B 0.000,C 90.000,E1 103.703} C_DIS
LIN {X 0.155,Y -654.170,Z 1243.373,A 0.000,B 0.000,C 90.000,E1 103.175} C_DIS
LIN {X -0.085,Y -654.834,Z 1243.371,A 0.000,B 0.000,C 90.000,E1 102.703} C_DIS
LIN {X -0.345,Y -655.105,Z 1243.369,A 0.000,B 0.000,C 90.000,E1 102.479} C_DIS
LIN {X 0.064,Y -655.266,Z 1243.366,A 0.000,B 0.000,C 90.000,E1 101.951} C_DIS
LIN {X -0.168,Y -655.073,Z 1243.364,A 0.000,B 0.000,C 90.000,E1 101.478} C_DIS
LIN {X -0.285,Y -654.900,Z 1243.362,A 0.000,B 0.000,C 90.000,E1 101.243} C_DIS
LIN {X 0.118,Y -654.276,Z 1243.360,A 0.000,B 0.000,C 90.000,E1 100.715} C_DIS
LIN {X -0.246,Y -653.321,Z 1243.357,A 0.000,B 0.000,C 90.000,E1 100.254} C_DIS
LIN {X 0.144,Y -652.063,Z 1243.354,A 0.000,B 0.000,C 90.000,E1 99.726} C_DIS
LIN {X -0.095,Y -651.331,Z 1243.353,A 0.000,B 0.000,C 90.000,E1 99.500} C_DIS
LIN {X 0.278,Y -649.532,Z 1243.350,A 0.000,B 0.000,C 90.000,E1 98.973} C_DIS
LIN {X -0.226,Y -646.678,Z 1243.347,A 0.000,B 0.000,C 90.000,E1 98.398} C_DIS
LIN {X 0.105,Y -644.108,Z 1243.344,A 0.000,B 0.000,C 90.000,E1 97.871} C_DIS
LIN {X 0.323,Y -641.120,Z 1243.341,A 0.000,B 0.000,C 90.000,E1 97.352} C_DIS
LIN {X -0.241,Y -636.772,Z 1243.338,A 0.000,B 0.000,C 90.000,E1 96.777} C_DIS
LIN {X -0.068,Y -632.959,Z 1243.335,A 0.000,B 0.000,C 90.000,E1 96.258} C_DIS
LIN {X 0.078,Y -628.551,Z 1243.332,A 0.000,B 0.000,C 90.000,E1 95.739} C_DIS
LIN {X 0.219,Y -623.687,Z 1243.329,A 0.000,B 0.000,C 90.000,E1 95.220} C_DIS
LIN {X -0.188,Y -617.135,Z 1243.326,A 0.000,B 0.000,C 90.000,E1 94.645} C_DIS
LIN {X -0.193,Y -610.099,Z 1243.323,A 0.000,B 0.000,C 90.000,E1 94.073} C_DIS
LIN {X 0.188,Y -602.486,Z 1243.320,A 0.000,B 0.000,C 90.000,E1 93.498} C_DIS
LIN {X -0.178,Y -594.631,Z 1243.317,A 0.000,B 0.000,C 90.000,E1 93.037} C_DIS
LIN {X 0.037,Y -584.936,Z 1243.314,A 0.000,B 0.000,C 90.000,E1 92.465} C_DIS
LIN {X -0.290,Y -583.259,Z 1243.313,A 0.000,B 0.000,C 90.000,E1 92.407} C_DIS
LIN {X -0.166,Y -570.863,Z 1243.310,A 0.000,B 0.000,C 90.000,E1 91.892} C_DIS
LIN {X -0.003,Y -567.203,Z 1243.309,A 0.000,B 0.000,C 90.000,E1 91.661} C_DIS
LIN {X -0.046,Y -567.141,Z 1243.309,A 0.000,B 0.000,C 90.000,E1 91.661} C_DIS
LIN {X -0.086,Y -566.927,Z 1243.309,A 0.000,B 0.000,C 90.000,E1 91.604} C_DIS
LIN {X 0.217,Y -566.384,Z 1243.307,A 0.000,B 0.000,C 90.000,E1 91.260} C_DIS
LIN {X -0.116,Y -566.347,Z 1243.304,A 0.000,B 0.000,C 90.000,E1 90.745} C_DIS
LIN {X 0.142,Y -567.712,Z 1243.293,A 0.000,B 0.000,C 90.000,E1 88.797} C_DIS
LIN {X -0.249,Y -568.939,Z 1243.284,A 0.000,B 0.000,C 90.000,E1 87.192} C_DIS
LIN {X -0.173,Y -571.139,Z 1243.271,A 0.000,B 0.000,C 90.000,E1 84.723} C_DIS
LIN {X 0.158,Y -572.747,Z 1243.262,A 0.000,B 0.000,C 90.000,E1 83.053} C_DIS
LIN {X 0.024,Y -574.427,Z 1243.252,A 0.000,B 0.000,C 90.000,E1 81.432} C_DIS
LIN {X -0.188,Y -575.698,Z 1243.245,A 0.000,B 0.000,C 90.000,E1 80.095} C_DIS
LIN {X -0.025,Y -576.490,Z 1243.239,A 0.000,B 0.000,C 90.000,E1 78.993} C_DIS
LIN {X -0.096,Y -577.436,Z 1243.231,A 0.000,B 0.000,C 90.000,E1 77.645} C_DIS
LIN {X 0.197,Y -578.204,Z 1243.225,A 0.000,B 0.000,C 90.000,E1 76.533} C_DIS
LIN {X -0.271,Y -579.063,Z 1243.218,A 0.000,B 0.000,C 90.000,E1 75.227} C_DIS
LIN {X 0.213,Y -579.952,Z 1243.209,A 0.000,B 0.000,C 90.000,E1 73.559} C_DIS
LIN {X 0.116,Y -580.570,Z 1243.203,A 0.000,B 0.000,C 90.000,E1 72.489} C_DIS
LIN {X 0.243,Y -581.586,Z 1243.194,A 0.000,B 0.000,C 90.000,E1 70.859} C_DIS
LIN {X -0.211,Y -582.189,Z 1243.188,A 0.000,B 0.000,C 90.000,E1 69.826} C_DIS
LIN {X -0.135,Y -583.586,Z 1243.176,A 0.000,B 0.000,C 90.000,E1 67.667} C_DIS
LIN {X -0.071,Y -584.858,Z 1243.167,A 0.000,B 0.000,C 90.000,E1 66.049} C_DIS
LIN {X -0.034,Y -585.821,Z 1243.161,A 0.000,B 0.000,C 90.000,E1 64.973} C_DIS
LIN {X 0.233,Y -587.987,Z 1243.148,A 0.000,B 0.000,C 90.000,E1 62.538} C_DIS
LIN {X -0.153,Y -589.623,Z 1243.139,A 0.000,B 0.000,C 90.000,E1 60.973} C_DIS
LIN {X 0.293,Y -591.285,Z 1243.130,A 0.000,B 0.000,C 90.000,E1 59.331} C_DIS
LIN {X 0.160,Y -592.389,Z 1243.124,A 0.000,B 0.000,C 90.000,E1 58.280} C_DIS
LIN {X 0.060,Y -593.670,Z 1243.117,A 0.000,B 0.000,C 90.000,E1 56.962} C_DIS
LIN {X -0.120,Y -595.097,Z 1243.108,A 0.000,B 0.000,C 90.000,E1 55.388} C_DIS
LIN {X 0.057,Y -596.472,Z 1243.099,A 0.000,B 0.000,C 90.000,E1 53.783} C_DIS
LIN {X 0.134,Y -597.671,Z 1243.090,A 0.000,B 0.000,C 90.000,E1 52.190} C_DIS
LIN {X -0.236,Y -598.518,Z 1243.084,A 0.000,B 0.000,C 90.000,E1 51.170} C_DIS
LIN {X 0.009,Y -598.944,Z 1243.080,A 0.000,B 0.000,C 90.000,E1 50.356} C_DIS
LIN {X 0.271,Y -599.614,Z 1243.073,A 0.000,B 0.000,C 90.000,E1 49.013} C_DIS
LIN {X -0.125,Y -600.295,Z 1243.064,A 0.000,B 0.000,C 90.000,E1 47.472} C_DIS
LIN {X 0.108,Y -600.533,Z 1243.056,A 0.000,B 0.000,C 90.000,E1 46.134} C_DIS
LIN {X 0.332,Y -600.619,Z 1243.052,A 0.000,B 0.000,C 90.000,E1 45.324} C_DIS
LIN {X 0.349,Y -600.562,Z 1243.046,A 0.000,B 0.000,C 90.000,E1 44.271} C_DIS
LIN {X -0.261,Y -600.275,Z 1243.039,A 0.000,B 0.000,C 90.000,E1 43.014} C_DIS
LIN {X -0.048,Y -600.007,Z 1243.035,A 0.000,B 0.000,C 90.000,E1 42.204} C_DIS
LIN {X 0.204,Y -599.648,Z 1243.030,A 0.000,B 0.000,C 90.000,E1 41.391} C_DIS
LIN {X 0.021,Y -599.007,Z 1243.023,A 0.000,B 0.000,C 90.000,E1 40.092} C_DIS
LIN {X 0.270,Y -598.564,Z 1243.018,A 0.000,B 0.000,C 90.000,E1 39.277} C_DIS
LIN {X -0.088,Y -597.704,Z 1243.013,A 0.000,B 0.000,C 90.000,E1 38.257} C_DIS
LIN {X 0.379,Y -596.721,Z 1243.007,A 0.000,B 0.000,C 90.000,E1 37.156} C_DIS
LIN {X 0.238,Y -595.819,Z 1243.002,A 0.000,B 0.000,C 90.000,E1 36.377} C_DIS
LIN {X 0.090,Y -594.707,Z 1242.998,A 0.000,B 0.000,C 90.000,E1 35.598} C_DIS
LIN {X 0.149,Y -592.982,Z 1242.992,A 0.000,B 0.000,C 90.000,E1 34.532} C_DIS
LIN {X -0.158,Y -590.909,Z 1242.986,A 0.000,B 0.000,C 90.000,E1 33.499} C_DIS
LIN {X 0.047,Y -590.360,Z 1242.985,A 0.000,B 0.000,C 90.000,E1 33.214} C_DIS
LIN {X 0.006,Y -588.321,Z 1242.980,A 0.000,B 0.000,C 90.000,E1 32.418} C_DIS
LIN {X 0.260,Y -586.035,Z 1242.976,A 0.000,B 0.000,C 90.000,E1 31.592} C_DIS
LIN {X 0.181,Y -583.439,Z 1242.971,A 0.000,B 0.000,C 90.000,E1 30.797} C_DIS
LIN {X 0.077,Y -580.361,Z 1242.967,A 0.000,B 0.000,C 90.000,E1 30.001} C_DIS
LIN {X 0.013,Y -577.524,Z 1242.963,A 0.000,B 0.000,C 90.000,E1 29.333} C_DIS
LIN {X -0.283,Y -574.936,Z 1242.960,A 0.000,B 0.000,C 90.000,E1 28.821} C_DIS
LIN {X -0.058,Y -570.098,Z 1242.955,A 0.000,B 0.000,C 90.000,E1 27.847} C_DIS
LIN {X 0.278,Y -566.131,Z 1242.951,A 0.000,B 0.000,C 90.000,E1 27.129} C_DIS
LIN {X -0.180,Y -561.879,Z 1242.947,A 0.000,B 0.000,C 90.000,E1 26.488} C_DIS
LIN {X -0.068,Y -558.267,Z 1242.944,A 0.000,B 0.000,C 90.000,E1 25.924} C_DIS
LIN {X 0.150,Y -553.379,Z 1242.940,A 0.000,B 0.000,C 90.000,E1 25.207} C_DIS
LIN {X 0.200,Y -549.177,Z 1242.937,A 0.000,B 0.000,C 90.000,E1 24.643} C_DIS
LIN {X 0.098,Y -543.579,Z 1242.933,A 0.000,B 0.000,C 90.000,E1 23.951} C_DIS
LIN {X -0.050,Y -537.415,Z 1242.929,A 0.000,B 0.000,C 90.000,E1 23.259} C_DIS
LIN {X 0.119,Y -529.839,Z 1242.924,A 0.000,B 0.000,C 90.000,E1 22.386} C_DIS
LIN {X 0.260,Y -520.646,Z 1242.919,A 0.000,B 0.000,C 90.000,E1 21.408} C_DIS
LIN {X -0.022,Y -512.527,Z 1242.915,A 0.000,B 0.000,C 90.000,E1 20.610} C_DIS
LIN {X 0.180,Y -508.370,Z 1242.912,A 0.000,B 0.000,C 90.000,E1 20.174} C_DIS
LIN {X -0.245,Y -498.577,Z 1242.907,A 0.000,B 0.000,C 90.000,E1 19.268} C_DIS
LIN {X -0.125,Y -487.055,Z 1242.901,A 0.000,B 0.000,C 90.000,E1 18.181} C_DIS
LIN {X -0.035,Y -479.647,Z 1242.897,A 0.000,B 0.000,C 90.000,E1 17.511} C_DIS
LIN {X -0.047,Y -464.869,Z 1242.890,A 0.000,B 0.000,C 90.000,E1 16.205} C_DIS
LIN {X -0.065,Y -447.109,Z 1242.881,A 0.000,B 0.000,C 90.000,E1 14.592} C_DIS
LIN {X 0.120,Y -426.919,Z 1242.870,A 0.000,B 0.000,C 90.000,E1 12.591} C_DIS
LIN {X -0.038,Y -404.237,Z 1242.856,A 0.000,B 0.000,C 90.000,E1 10.141} C_DIS
LIN {X -0.142,Y -400.139,Z 1242.854,A 0.000,B 0.000,C 90.000,E1 9.670} C_DIS
LIN {X 0.026,Y -396.943,Z 1242.851,A 0.000,B 0.000,C 90.000,E1 9.208} C_DIS
LIN {X 0.050,Y -395.840,Z 1242.850,A 0.000,B 0.000,C 90.000,E1 9.029} C_DIS
LIN {X -0.069,Y -394.462,Z 1242.849,A 0.000,B 0.000,C 90.000,E1 8.746} C_DIS
LIN {X -0.107,Y -394.454,Z 1242.849,A 0.000,B 0.000,C 90.000,E1 8.746} C_DIS
LIN {X 0.060,Y -394.337,Z 1242.848,A 0.000,B 0.000,C 90.000,E1 8.568} C_DIS
LIN {X 0.022,Y -394.332,Z 1242.848,A 0.000,B 0.000,C 90.000,E1 8.568} C_DIS
LIN {X -0.031,Y -396.391,Z 1242.845,A 0.000,B 0.000,C 90.000,E1 8.106} C_DIS
LIN {X -0.040,Y -400.767,Z 1242.843,A 0.000,B 0.000,C 90.000,E1 7.644} C_DIS
LIN {X -0.008,Y -406.120,Z 1242.840,A 0.000,B 0.000,C 90.000,E1 7.239} C_DIS
LIN {X -0.174,Y -413.955,Z 1242.837,A 0.000,B 0.000,C 90.000,E1 6.720} C_DIS
LIN {X -0.136,Y -425.038,Z 1242.833,A 0.000,B 0.000,C 90.000,E1 5.910} C_DIS
LIN {X 0.200,Y -431.338,Z 1242.830,A 0.000,B 0.000,C 90.000,E1 5.391} C_DIS
LIN {X 0.139,Y -442.379,Z 1242.825,A 0.000,B 0.000,C 90.000,E1 4.531} C_DIS
LIN {X -0.152,Y -451.528,Z 1242.821,A 0.000,B 0.000,C 90.000,E1 3.841} C_DIS
LIN {X -0.112,Y -462.086,Z 1242.817,A 0.000,B 0.000,C 90.000,E1 2.980} C_DIS
LIN {X -0.023,Y -468.096,Z 1242.814,A 0.000,B 0.000,C 90.000,E1 2.465} C_DIS
LIN {X -0.054,Y -473.909,Z 1242.811,A 0.000,B 0.000,C 90.000,E1 1.949} C_DIS
LIN {X -0.023,Y -479.388,Z 1242.808,A 0.000,B 0.000,C 90.000,E1 1.432} C_DIS
LIN {X 0.015,Y -485.977,Z 1242.804,A 0.000,B 0.000,C 90.000,E1 0.745} C_DIS
LIN {X 0.128,Y -492.486,Z 1242.800,A 0.000,B 0.000,C 90.000,E1 360.000} C_DIS
LIN {X 0.209,Y -496.834,Z 1242.797,A 0.000,B 0.000,C 90.000,E1 359.484} C_DIS
LIN {X 0.129,Y -502.648,Z 1242.793,A 0.000,B 0.000,C 90.000,E1 358.740} C_DIS
LIN {X 0.113,Y -508.021,Z 1242.789,A 0.000,B 0.000,C 90.000,E1 357.993} C_DIS
LIN {X 0.131,Y -512.966,Z 1242.785,A 0.000,B 0.000,C 90.000,E1 357.249} C_DIS
LIN {X 0.217,Y -517.690,Z 1242.781,A 0.000,B 0.000,C 90.000,E1 356.502} C_DIS
LIN {X 0.120,Y -521.202,Z 1242.777,A 0.000,B 0.000,C 90.000,E1 355.927} C_DIS
LIN {X -0.277,Y -525.173,Z 1242.773,A 0.000,B 0.000,C 90.000,E1 355.241} C_DIS
LIN {X -0.031,Y -528.802,Z 1242.769,A 0.000,B 0.000,C 90.000,E1 354.489} C_DIS
LIN {X -0.045,Y -531.526,Z 1242.766,A 0.000,B 0.000,C 90.000,E1 353.913} C_DIS
LIN {X -0.040,Y -534.081,Z 1242.763,A 0.000,B 0.000,C 90.000,E1 353.337} C_DIS
LIN {X -0.020,Y -536.451,Z 1242.760,A 0.000,B 0.000,C 90.000,E1 352.761} C_DIS
LIN {X 0.073,Y -539.665,Z 1242.755,A 0.000,B 0.000,C 90.000,E1 351.894} C_DIS
LIN {X 0.199,Y -542.578,Z 1242.750,A 0.000,B 0.000,C 90.000,E1 351.027} C_DIS
LIN {X -0.093,Y -545.330,Z 1242.746,A 0.000,B 0.000,C 90.000,E1 350.208} C_DIS
LIN {X 0.187,Y -548.540,Z 1242.739,A 0.000,B 0.000,C 90.000,E1 349.050} C_DIS
LIN {X 0.187,Y -552.131,Z 1242.732,A 0.000,B 0.000,C 90.000,E1 347.645} C_DIS
LIN {X -0.165,Y -555.247,Z 1242.724,A 0.000,B 0.000,C 90.000,E1 346.284} C_DIS
LIN {X -0.192,Y -557.432,Z 1242.718,A 0.000,B 0.000,C 90.000,E1 345.172} C_DIS
LIN {X -0.189,Y -558.922,Z 1242.713,A 0.000,B 0.000,C 90.000,E1 344.338} C_DIS
LIN {X 0.127,Y -560.755,Z 1242.707,A 0.000,B 0.000,C 90.000,E1 343.196} C_DIS
LIN {X 0.077,Y -562.557,Z 1242.699,A 0.000,B 0.000,C 90.000,E1 341.819} C_DIS
LIN {X -0.088,Y -563.695,Z 1242.693,A 0.000,B 0.000,C 90.000,E1 340.732} C_DIS
LIN {X -0.047,Y -564.401,Z 1242.687,A 0.000,B 0.000,C 90.000,E1 339.625} C_DIS
LIN {X -0.121,Y -564.606,Z 1242.684,A 0.000,B 0.000,C 90.000,E1 339.082} C_DIS
LIN {X -0.198,Y -564.686,Z 1242.681,A 0.000,B 0.000,C 90.000,E1 338.539} C_DIS
LIN {X 0.261,Y -564.445,Z 1242.676,A 0.000,B 0.000,C 90.000,E1 337.667} C_DIS
LIN {X -0.126,Y -564.181,Z 1242.673,A 0.000,B 0.000,C 90.000,E1 337.155} C_DIS
LIN {X 0.108,Y -563.318,Z 1242.668,A 0.000,B 0.000,C 90.000,E1 336.305} C_DIS
LIN {X 0.038,Y -562.333,Z 1242.664,A 0.000,B 0.000,C 90.000,E1 335.485} C_DIS
LIN {X 0.155,Y -561.429,Z 1242.661,A 0.000,B 0.000,C 90.000,E1 334.921} C_DIS
LIN {X 0.063,Y -559.740,Z 1242.656,A 0.000,B 0.000,C 90.000,E1 334.101} C_DIS
LIN {X 0.201,Y -557.893,Z 1242.652,A 0.000,B 0.000,C 90.000,E1 333.256} C_DIS
LIN {X 0.066,Y -555.465,Z 1242.647,A 0.000,B 0.000,C 90.000,E1 332.436} C_DIS
LIN {X 0.159,Y -552.745,Z 1242.642,A 0.000,B 0.000,C 90.000,E1 331.591} C_DIS
LIN {X -0.259,Y -549.333,Z 1242.638,A 0.000,B 0.000,C 90.000,E1 330.795} C_DIS
LIN {X 0.037,Y -545.264,Z 1242.633,A 0.000,B 0.000,C 90.000,E1 329.921} C_DIS
LIN {X 0.143,Y -541.328,Z 1242.629,A 0.000,B 0.000,C 90.000,E1 329.203} C_DIS
LIN {X -0.251,Y -536.821,Z 1242.625,A 0.000,B 0.000,C 90.000,E1 328.535} C_DIS
LIN {X -0.095,Y -531.078,Z 1242.620,A 0.000,B 0.000,C 90.000,E1 327.661} C_DIS
LIN {X -0.009,Y -524.907,Z 1242.615,A 0.000,B 0.000,C 90.000,E1 326.786} C_DIS
LIN {X 0.276,Y -516.576,Z 1242.609,A 0.000,B 0.000,C 90.000,E1 325.595} C_DIS
LIN {X -0.151,Y -512.873,Z 1242.606,A 0.000,B 0.000,C 90.000,E1 325.055} C_DIS
LIN {X -0.227,Y -511.161,Z 1242.604,A 0.000,B 0.000,C 90.000,E1 324.769} C_DIS
LIN {X 0.018,Y -508.580,Z 1242.601,A 0.000,B 0.000,C 90.000,E1 324.149} C_DIS
LIN {X -0.225,Y -507.082,Z 1242.598,A 0.000,B 0.000,C 90.000,E1 323.623} C_DIS
LIN {X -0.013,Y -505.918,Z 1242.594,A 0.000,B 0.000,C 90.000,E1 323.004} C_DIS
LIN {X 0.090,Y -505.174,Z 1242.591,A 0.000,B 0.000,C 90.000,E1 322.396} C_DIS
LIN {X -0.118,Y -504.782,Z 1242.588,A 0.000,B 0.000,C 90.000,E1 321.823} C_DIS
LIN {X -0.017,Y -504.658,Z 1242.585,A 0.000,B 0.000,C 90.000,E1 321.215} C_DIS
LIN {X -0.346,Y -505.291,Z 1242.575,A 0.000,B 0.000,C 90.000,E1 319.461} C_DIS
LIN {X 0.098,Y -505.858,Z 1242.566,A 0.000,B 0.000,C 90.000,E1 317.919} C_DIS
LIN {X 0.297,Y -506.544,Z 1242.555,A 0.000,B 0.000,C 90.000,E1 315.810} C_DIS
LIN {X 0.264,Y -506.988,Z 1242.545,A 0.000,B 0.000,C 90.000,E1 314.028} C_DIS
LIN {X -0.226,Y -507.665,Z 1242.533,A 0.000,B 0.000,C 90.000,E1 312.000} C_DIS
LIN {X 0.032,Y -508.097,Z 1242.527,A 0.000,B 0.000,C 90.000,E1 310.782} C_DIS
LIN {X 0.198,Y -508.490,Z 1242.518,A 0.000,B 0.000,C 90.000,E1 309.277} C_DIS
LIN {X -0.047,Y -509.007,Z 1242.508,A 0.000,B 0.000,C 90.000,E1 307.523} C_DIS
LIN {X 0.301,Y -509.322,Z 1242.502,A 0.000,B 0.000,C 90.000,E1 306.297} C_DIS
LIN {X 0.261,Y -509.604,Z 1242.494,A 0.000,B 0.000,C 90.000,E1 304.818} C_DIS
LIN {X -0.063,Y -509.858,Z 1242.485,A 0.000,B 0.000,C 90.000,E1 303.372} C_DIS
LIN {X -0.053,Y -510.036,Z 1242.476,A 0.000,B 0.000,C 90.000,E1 301.592} C_DIS
LIN {X -0.238,Y -510.067,Z 1242.464,A 0.000,B 0.000,C 90.000,E1 299.539} C_DIS
LIN {X 0.137,Y -509.984,Z 1242.454,A 0.000,B 0.000,C 90.000,E1 297.719} C_DIS
LIN {X -0.180,Y -509.887,Z 1242.444,A 0.000,B 0.000,C 90.000,E1 295.976} C_DIS
LIN {X -0.158,Y -510.101,Z 1242.433,A 0.000,B 0.000,C 90.000,E1 293.898} C_DIS
LIN {X 0.006,Y -510.000,Z 1242.426,A 0.000,B 0.000,C 90.000,E1 292.695} C_DIS
LIN {X -0.228,Y -509.620,Z 1242.420,A 0.000,B 0.000,C 90.000,E1 291.535} C_DIS
LIN {X -0.247,Y -508.817,Z 1242.410,A 0.000,B 0.000,C 90.000,E1 289.758} C_DIS
LIN {X 0.087,Y -508.198,Z 1242.401,A 0.000,B 0.000,C 90.000,E1 288.236} C_DIS
LIN {X 0.154,Y -507.729,Z 1242.395,A 0.000,B 0.000,C 90.000,E1 287.040} C_DIS
LIN {X 0.216,Y -507.311,Z 1242.388,A 0.000,B 0.000,C 90.000,E1 285.843} C_DIS
LIN {X 0.211,Y -506.562,Z 1242.380,A 0.000,B 0.000,C 90.000,E1 284.356} C_DIS
LIN {X 0.010,Y -505.370,Z 1242.370,A 0.000,B 0.000,C 90.000,E1 282.591} C_DIS
LIN {X -0.208,Y -504.457,Z 1242.363,A 0.000,B 0.000,C 90.000,E1 281.422} C_DIS
LIN {X -0.065,Y -503.176,Z 1242.353,A 0.000,B 0.000,C 90.000,E1 279.613} C_DIS
LIN {X 0.037,Y -501.250,Z 1242.337,A 0.000,B 0.000,C 90.000,E1 276.606} C_DIS
LIN {X -0.101,Y -500.293,Z 1242.327,A 0.000,B 0.000,C 90.000,E1 274.821} C_DIS
LIN {X 0.098,Y -499.124,Z 1242.315,A 0.000,B 0.000,C 90.000,E1 272.694} C_DIS
LIN {X -0.161,Y -497.683,Z 1242.305,A 0.000,B 0.000,C 90.000,E1 270.917} C_DIS
LIN {X 0.039,Y -496.465,Z 1242.295,A 0.000,B 0.000,C 90.000,E1 269.083} C_DIS
LIN {X 0.075,Y -495.192,Z 1242.283,A 0.000,B 0.000,C 90.000,E1 266.963} C_DIS
LIN {X 0.132,Y -493.982,Z 1242.271,A 0.000,B 0.000,C 90.000,E1 264.837} C_DIS
LIN {X -0.012,Y -492.990,Z 1242.263,A 0.000,B 0.000,C 90.000,E1 263.337} C_DIS
LIN {X -0.176,Y -491.750,Z 1242.255,A 0.000,B 0.000,C 90.000,E1 261.837} C_DIS
LIN {X 0.076,Y -489.941,Z 1242.244,A 0.000,B 0.000,C 90.000,E1 259.982} C_DIS
LIN {X 0.005,Y -487.475,Z 1242.228,A 0.000,B 0.000,C 90.000,E1 256.937} C_DIS
LIN {X -0.268,Y -485.960,Z 1242.214,A 0.000,B 0.000,C 90.000,E1 254.519} C_DIS
LIN {X -0.064,Y -485.232,Z 1242.207,A 0.000,B 0.000,C 90.000,E1 253.268} C_DIS
LIN {X 0.135,Y -484.049,Z 1242.195,A 0.000,B 0.000,C 90.000,E1 251.094} C_DIS
LIN {X 0.003,Y -483.267,Z 1242.187,A 0.000,B 0.000,C 90.000,E1 249.571} C_DIS
LIN {X 0.030,Y -482.486,Z 1242.178,A 0.000,B 0.000,C 90.000,E1 248.028} C_DIS
LIN {X 0.039,Y -481.572,Z 1242.169,A 0.000,B 0.000,C 90.000,E1 246.485} C_DIS
LIN {X 0.221,Y -480.736,Z 1242.163,A 0.000,B 0.000,C 90.000,E1 245.229} C_DIS
LIN {X 0.116,Y -479.144,Z 1242.151,A 0.000,B 0.000,C 90.000,E1 243.076} C_DIS
LIN {X 0.232,Y -477.926,Z 1242.142,A 0.000,B 0.000,C 90.000,E1 241.513} C_DIS
LIN {X -0.088,Y -476.587,Z 1242.133,A 0.000,B 0.000,C 90.000,E1 239.999} C_DIS
LIN {X 0.181,Y -474.487,Z 1242.121,A 0.000,B 0.000,C 90.000,E1 237.788} C_DIS
LIN {X -0.066,Y -473.673,Z 1242.116,A 0.000,B 0.000,C 90.000,E1 236.882} C_DIS
LIN {X 0.144,Y -471.457,Z 1242.102,A 0.000,B 0.000,C 90.000,E1 234.356} C_DIS
LIN {X 0.047,Y -469.575,Z 1242.088,A 0.000,B 0.000,C 90.000,E1 231.859} C_DIS
LIN {X -0.020,Y -467.795,Z 1242.076,A 0.000,B 0.000,C 90.000,E1 229.666} C_DIS
LIN {X 0.058,Y -466.621,Z 1242.067,A 0.000,B 0.000,C 90.000,E1 228.081} C_DIS
LIN {X -0.177,Y -465.228,Z 1242.057,A 0.000,B 0.000,C 90.000,E1 226.215} C_DIS
LIN {X 0.175,Y -463.637,Z 1242.037,A 0.000,B 0.000,C 90.000,E1 222.690} C_DIS
LIN {X 0.113,Y -464.827,Z 1241.999,A 0.000,B 0.000,C 90.000,E1 215.724} C_DIS
LIN {X -0.177,Y -468.129,Z 1241.974,A 0.000,B 0.000,C 90.000,E1 211.337} C_DIS
LIN {X 0.099,Y -471.924,Z 1241.955,A 0.000,B 0.000,C 90.000,E1 207.847} C_DIS
LIN {X 0.089,Y -473.860,Z 1241.946,A 0.000,B 0.000,C 90.000,E1 206.283} C_DIS
LIN {X -0.228,Y -478.114,Z 1241.929,A 0.000,B 0.000,C 90.000,E1 203.206} C_DIS
LIN {X 0.150,Y -483.296,Z 1241.912,A 0.000,B 0.000,C 90.000,E1 200.066} C_DIS
LIN {X -0.214,Y -489.485,Z 1241.895,A 0.000,B 0.000,C 90.000,E1 197.040} C_DIS
LIN {X -0.030,Y -493.722,Z 1241.884,A 0.000,B 0.000,C 90.000,E1 195.190} C_DIS
LIN {X 0.122,Y -497.964,Z 1241.874,A 0.000,B 0.000,C 90.000,E1 193.355} C_DIS
LIN {X -0.093,Y -500.867,Z 1241.868,A 0.000,B 0.000,C 90.000,E1 192.175} C_DIS
LIN {X -0.006,Y -505.409,Z 1241.858,A 0.000,B 0.000,C 90.000,E1 190.366} C_DIS
LIN {X 0.055,Y -510.854,Z 1241.846,A 0.000,B 0.000,C 90.000,E1 188.276} C_DIS
LIN {X 0.242,Y -514.789,Z 1241.838,A 0.000,B 0.000,C 90.000,E1 186.777} C_DIS
LIN {X -0.011,Y -518.621,Z 1241.830,A 0.000,B 0.000,C 90.000,E1 185.334} C_DIS
LIN {X 0.220,Y -523.235,Z 1241.820,A 0.000,B 0.000,C 90.000,E1 183.555} C_DIS
LIN {X -0.003,Y -528.514,Z 1241.809,A 0.000,B 0.000,C 90.000,E1 181.547} C_DIS
LIN {X -0.125,Y -533.657,Z 1241.797,A 0.000,B 0.000,C 90.000,E1 179.542} C_DIS
LIN {X -0.119,Y -537.209,Z 1241.789,A 0.000,B 0.000,C 90.000,E1 178.108} C_DIS
LIN {X -0.045,Y -540.532,Z 1241.781,A 0.000,B 0.000,C 90.000,E1 176.674} C_DIS
LIN {X 0.040,Y -542.420,Z 1241.777,A 0.000,B 0.000,C 90.000,E1 175.812} C_DIS
LIN {X -0.278,Y -546.136,Z 1241.767,A 0.000,B 0.000,C 90.000,E1 174.147} C_DIS
LIN {X -0.056,Y -548.480,Z 1241.761,A 0.000,B 0.000,C 90.000,E1 172.996} C_DIS
LIN {X -0.170,Y -551.251,Z 1241.753,A 0.000,B 0.000,C 90.000,E1 171.602} C_DIS
LIN {X -0.194,Y -554.458,Z 1241.744,A 0.000,B 0.000,C 90.000,E1 169.926} C_DIS
LIN {X -0.097,Y -556.996,Z 1241.736,A 0.000,B 0.000,C 90.000,E1 168.522} C_DIS
LIN {X 0.193,Y -560.018,Z 1241.727,A 0.000,B 0.000,C 90.000,E1 166.825} C_DIS
LIN {X 0.127,Y -563.077,Z 1241.718,A 0.000,B 0.000,C 90.000,E1 165.172} C_DIS
LIN {X 0.161,Y -568.786,Z 1241.703,A 0.000,B 0.000,C 90.000,E1 162.417} C_DIS
LIN {X 0.070,Y -573.316,Z 1241.693,A 0.000,B 0.000,C 90.000,E1 160.786} C_DIS
LIN {X -0.108,Y -577.977,Z 1241.686,A 0.000,B 0.000,C 90.000,E1 159.444} C_DIS
LIN {X 0.190,Y -584.466,Z 1241.677,A 0.000,B 0.000,C 90.000,E1 157.794} C_DIS
LIN {X 0.208,Y -592.931,Z 1241.666,A 0.000,B 0.000,C 90.000,E1 155.921} C_DIS
LIN {X 0.293,Y -599.130,Z 1241.659,A 0.000,B 0.000,C 90.000,E1 154.588} C_DIS
LIN {X -0.051,Y -605.159,Z 1241.652,A 0.000,B 0.000,C 90.000,E1 153.307} C_DIS
LIN {X 0.231,Y -610.965,Z 1241.645,A 0.000,B 0.000,C 90.000,E1 151.975} C_DIS
LIN {X -0.184,Y -616.490,Z 1241.637,A 0.000,B 0.000,C 90.000,E1 150.717} C_DIS
LIN {X 0.019,Y -622.975,Z 1241.629,A 0.000,B 0.000,C 90.000,E1 149.154} C_DIS
LIN {X 0.122,Y -628.127,Z 1241.622,A 0.000,B 0.000,C 90.000,E1 147.867} C_DIS
LIN {X 0.303,Y -632.203,Z 1241.616,A 0.000,B 0.000,C 90.000,E1 146.834} C_DIS
LIN {X 0.037,Y -636.856,Z 1241.609,A 0.000,B 0.000,C 90.000,E1 145.595} C_DIS
LIN {X -0.187,Y -640.398,Z 1241.603,A 0.000,B 0.000,C 90.000,E1 144.609} C_DIS
LIN {X 0.152,Y -643.603,Z 1241.598,A 0.000,B 0.000,C 90.000,E1 143.577} C_DIS
LIN {X -0.117,Y -646.508,Z 1241.592,A 0.000,B 0.000,C 90.000,E1 142.603} C_DIS
LIN {X 0.208,Y -649.961,Z 1241.585,A 0.000,B 0.000,C 90.000,E1 141.331} C_DIS
LIN {X 0.036,Y -652.478,Z 1241.580,A 0.000,B 0.000,C 90.000,E1 140.356} C_DIS
LIN {X 0.305,Y -656.162,Z 1241.572,A 0.000,B 0.000,C 90.000,E1 138.852} C_DIS
LIN {X 0.151,Y -659.719,Z 1241.563,A 0.000,B 0.000,C 90.000,E1 137.391} C_DIS
LIN {X -0.407,Y -662.567,Z 1241.557,A 0.000,B 0.000,C 90.000,E1 136.215} C_DIS
LIN {X 0.017,Y -668.765,Z 1241.543,A 0.000,B 0.000,C 90.000,E1 133.743} C_DIS
LIN {X 0.090,Y -673.158,Z 1241.534,A 0.000,B 0.000,C 90.000,E1 132.043} C_DIS
LIN {X -0.204,Y -676.333,Z 1241.527,A 0.000,B 0.000,C 90.000,E1 130.862} C_DIS
LIN {X 0.029,Y -680.107,Z 1241.519,A 0.000,B 0.000,C 90.000,E1 129.402} C_DIS
LIN {X 0.032,Y -684.387,Z 1241.510,A 0.000,B 0.000,C 90.000,E1 127.729} C_DIS
LIN {X 0.056,Y -687.420,Z 1241.503,A 0.000,B 0.000,C 90.000,E1 126.537} C_DIS
LIN {X 0.312,Y -689.131,Z 1241.499,A 0.000,B 0.000,C 90.000,E1 125.804} C_DIS
LIN {X 0.058,Y -692.301,Z 1241.491,A 0.000,B 0.000,C 90.000,E1 124.405} C_DIS
LIN {X -0.146,Y -695.412,Z 1241.483,A 0.000,B 0.000,C 90.000,E1 123.007} C_DIS
LIN {X 0.006,Y -697.317,Z 1241.478,A 0.000,B 0.000,C 90.000,E1 122.054} C_DIS
LIN {X -0.003,Y -700.417,Z 1241.469,A 0.000,B 0.000,C 90.000,E1 120.413} C_DIS
LIN {X -0.064,Y -701.658,Z 1241.465,A 0.000,B 0.000,C 90.000,E1 119.716} C_DIS
LIN {X -0.257,Y -703.463,Z 1241.459,A 0.000,B 0.000,C 90.000,E1 118.565} C_DIS
LIN {X -0.028,Y -704.323,Z 1241.455,A 0.000,B 0.000,C 90.000,E1 117.847} C_DIS
LIN {X -0.133,Y -705.229,Z 1241.450,A 0.000,B 0.000,C 90.000,E1 116.924} C_DIS
LIN {X -0.211,Y -705.614,Z 1241.446,A 0.000,B 0.000,C 90.000,E1 116.232} C_DIS
LIN {X 0.370,Y -705.745,Z 1241.443,A 0.000,B 0.000,C 90.000,E1 115.720} C_DIS
LIN {X 0.303,Y -705.535,Z 1241.439,A 0.000,B 0.000,C 90.000,E1 115.027} C_DIS
LIN {X -0.052,Y -705.179,Z 1241.437,A 0.000,B 0.000,C 90.000,E1 114.591} C_DIS
LIN {X -0.120,Y -704.398,Z 1241.434,A 0.000,B 0.000,C 90.000,E1 114.131} C_DIS
LIN {X -0.121,Y -703.826,Z 1241.433,A 0.000,B 0.000,C 90.000,E1 113.898} C_DIS
LIN {X -0.203,Y -701.890,Z 1241.430,A 0.000,B 0.000,C 90.000,E1 113.439} C_DIS
LIN {X -0.343,Y -701.279,Z 1241.430,A 0.000,B 0.000,C 90.000,E1 113.334} C_DIS
LIN {X -0.205,Y -700.350,Z 1241.429,A 0.000,B 0.000,C 90.000,E1 113.206} C_DIS
LIN {X 0.149,Y -695.570,Z 1241.426,A 0.000,B 0.000,C 90.000,E1 112.717} C_DIS
LIN {X 0.282,Y -693.841,Z 1241.426,A 0.000,B 0.000,C 90.000,E1 112.589} C_DIS
LIN {X -0.225,Y -690.802,Z 1241.425,A 0.000,B 0.000,C 90.000,E1 112.514} C_DIS
LIN {X 0.145,Y -686.203,Z 1241.424,A 0.000,B 0.000,C 90.000,E1 112.333} C_DIS
LIN {X -0.101,Y -685.186,Z 1241.424,A 0.000,B 0.000,C 90.000,E1 112.333} C_DIS
LIN {X -0.255,Y -677.152,Z 1241.424,A 0.000,B 0.000,C 90.000,E1 112.280} C_DIS
LIN {X -0.033,Y -622.326,Z 1241.424,A 0.000,B 0.000,C 90.000,E1 112.259} C_DIS
LIN {X 0.031,Y -618.924,Z 1241.422,A 0.000,B 0.000,C 90.000,E1 112.025} C_DIS
LIN {X -0.284,Y -617.800,Z 1241.422,A 0.000,B 0.000,C 90.000,E1 111.897} C_DIS
LIN {X 0.256,Y -617.796,Z 1241.422,A 0.000,B 0.000,C 90.000,E1 111.844} C_DIS
LIN {X 0.063,Y -617.742,Z 1241.420,A 0.000,B 0.000,C 90.000,E1 111.589} C_DIS
LIN {X -0.315,Y -620.140,Z 1241.417,A 0.000,B 0.000,C 90.000,E1 111.046} C_DIS
LIN {X -0.006,Y -624.249,Z 1241.412,A 0.000,B 0.000,C 90.000,E1 110.248} C_DIS
LIN {X -0.242,Y -627.412,Z 1241.409,A 0.000,B 0.000,C 90.000,E1 109.631} C_DIS
LIN {X -0.071,Y -631.329,Z 1241.404,A 0.000,B 0.000,C 90.000,E1 108.725} C_DIS
LIN {X 0.078,Y -641.737,Z 1241.391,A 0.000,B 0.000,C 90.000,E1 106.441} C_DIS
LIN {X -0.220,Y -644.966,Z 1241.387,A 0.000,B 0.000,C 90.000,E1 105.717} C_DIS
LIN {X -0.040,Y -647.793,Z 1241.383,A 0.000,B 0.000,C 90.000,E1 104.954} C_DIS
LIN {X -0.318,Y -649.423,Z 1241.380,A 0.000,B 0.000,C 90.000,E1 104.481} C_DIS
LIN {X 0.072,Y -651.312,Z 1241.376,A 0.000,B 0.000,C 90.000,E1 103.703} C_DIS
LIN {X -0.187,Y -652.362,Z 1241.373,A 0.000,B 0.000,C 90.000,E1 103.231} C_DIS
LIN {X -0.068,Y -653.311,Z 1241.369,A 0.000,B 0.000,C 90.000,E1 102.479} C_DIS
LIN {X -0.311,Y -653.492,Z 1241.367,A 0.000,B 0.000,C 90.000,E1 102.007} C_DIS
LIN {X 0.086,Y -653.308,Z 1241.364,A 0.000,B 0.000,C 90.000,E1 101.478} C_DIS
LIN {X -0.163,Y -652.831,Z 1241.361,A 0.000,B 0.000,C 90.000,E1 101.007} C_DIS
LIN {X 0.231,Y -652.538,Z 1241.360,A 0.000,B 0.000,C 90.000,E1 100.725} C_DIS
LIN {X -0.022,Y -651.581,Z 1241.357,A 0.000,B 0.000,C 90.000,E1 100.254} C_DIS
LIN {X 0.355,Y -650.293,Z 1241.354,A 0.000,B 0.000,C 90.000,E1 99.726} C_DIS
LIN {X 0.111,Y -649.519,Z 1241.353,A 0.000,B 0.000,C 90.000,E1 99.500} C_DIS
LIN {X -0.169,Y -647.692,Z 1241.350,A 0.000,B 0.000,C 90.000,E1 99.029} C_DIS
LIN {X -0.048,Y -644.849,Z 1241.347,A 0.000,B 0.000,C 90.000,E1 98.398} C_DIS
LIN {X 0.269,Y -642.270,Z 1241.344,A 0.000,B 0.000,C 90.000,E1 97.871} C_DIS
LIN {X -0.160,Y -639.206,Z 1241.341,A 0.000,B 0.000,C 90.000,E1 97.409} C_DIS
LIN {X 0.027,Y -635.794,Z 1241.338,A 0.000,B 0.000,C 90.000,E1 96.891} C_DIS
LIN {X 0.190,Y -631.977,Z 1241.336,A 0.000,B 0.000,C 90.000,E1 96.372} C_DIS
LIN {X 0.185,Y -626.485,Z 1241.332,A 0.000,B 0.000,C 90.000,E1 95.739} C_DIS
LIN {X -0.274,Y -621.421,Z 1241.329,A 0.000,B 0.000,C 90.000,E1 95.277} C_DIS
LIN {X 0.096,Y -617.547,Z 1241.327,A 0.000,B 0.000,C 90.000,E1 94.878} C_DIS
LIN {X 0.064,Y -610.582,Z 1241.324,A 0.000,B 0.000,C 90.000,E1 94.302} C_DIS
LIN {X 0.213,Y -606.035,Z 1241.322,A 0.000,B 0.000,C 90.000,E1 93.955} C_DIS
LIN {X 0.078,Y -599.984,Z 1241.320,A 0.000,B 0.000,C 90.000,E1 93.555} C_DIS
LIN {X 0.199,Y -593.717,Z 1241.318,A 0.000,B 0.000,C 90.000,E1 93.154} C_DIS
LIN {X -0.076,Y -587.254,Z 1241.316,A 0.000,B 0.000,C 90.000,E1 92.808} C_DIS
LIN {X 0.141,Y -582.238,Z 1241.314,A 0.000,B 0.000,C 90.000,E1 92.522} C_DIS
LIN {X 0.095,Y -576.597,Z 1241.313,A 0.000,B 0.000,C 90.000,E1 92.293} C_DIS
LIN {X -0.217,Y -571.514,Z 1241.312,A 0.000,B 0.000,C 90.000,E1 92.121} C_DIS
LIN {X 0.246,Y -570.080,Z 1241.311,A 0.000,B 0.000,C 90.000,E1 92.007} C_DIS
LIN {X 0.077,Y -567.165,Z 1241.310,A 0.000,B 0.000,C 90.000,E1 91.835} C_DIS
LIN {X -0.224,Y -566.650,Z 1241.310,A 0.000,B 0.000,C 90.000,E1 91.776} C_DIS
LIN {X -0.265,Y -566.636,Z 1241.310,A 0.000,B 0.000,C 90.000,E1 91.776} C_DIS
LIN {X 0.063,Y -566.499,Z 1241.308,A 0.000,B 0.000,C 90.000,E1 91.489} C_DIS
LIN {X 0.179,Y -566.140,Z 1241.307,A 0.000,B 0.000,C 90.000,E1 91.203} C_DIS
LIN {X 0.144,Y -566.627,Z 1241.301,A 0.000,B 0.000,C 90.000,E1 90.229} C_DIS
LIN {X 0.168,Y -567.621,Z 1241.294,A 0.000,B 0.000,C 90.000,E1 88.854} C_DIS
LIN {X -0.225,Y -568.862,Z 1241.285,A 0.000,B 0.000,C 90.000,E1 87.249} C_DIS
LIN {X 0.025,Y -571.267,Z 1241.269,A 0.000,B 0.000,C 90.000,E1 84.489} C_DIS
LIN {X -0.202,Y -572.880,Z 1241.260,A 0.000,B 0.000,C 90.000,E1 82.875} C_DIS
LIN {X 0.244,Y -574.531,Z 1241.251,A 0.000,B 0.000,C 90.000,E1 81.197} C_DIS
LIN {X -0.169,Y -575.539,Z 1241.245,A 0.000,B 0.000,C 90.000,E1 80.151} C_DIS
LIN {X -0.005,Y -576.341,Z 1241.239,A 0.000,B 0.000,C 90.000,E1 79.050} C_DIS
LIN {X 0.275,Y -577.080,Z 1241.233,A 0.000,B 0.000,C 90.000,E1 77.937} C_DIS
LIN {X -0.131,Y -578.174,Z 1241.224,A 0.000,B 0.000,C 90.000,E1 76.353} C_DIS
LIN {X -0.036,Y -579.015,Z 1241.217,A 0.000,B 0.000,C 90.000,E1 74.991} C_DIS
LIN {X 0.100,Y -580.093,Z 1241.206,A 0.000,B 0.000,C 90.000,E1 73.087} C_DIS
LIN {X -0.083,Y -581.547,Z 1241.193,A 0.000,B 0.000,C 90.000,E1 70.678} C_DIS
LIN {X 0.210,Y -582.125,Z 1241.187,A 0.000,B 0.000,C 90.000,E1 69.571} C_DIS
LIN {X -0.063,Y -583.803,Z 1241.173,A 0.000,B 0.000,C 90.000,E1 67.177} C_DIS
LIN {X 0.116,Y -585.402,Z 1241.163,A 0.000,B 0.000,C 90.000,E1 65.281} C_DIS
LIN {X 0.111,Y -587.564,Z 1241.149,A 0.000,B 0.000,C 90.000,E1 62.871} C_DIS
LIN {X 0.114,Y -589.437,Z 1241.139,A 0.000,B 0.000,C 90.000,E1 61.001} C_DIS
LIN {X 0.035,Y -591.095,Z 1241.130,A 0.000,B 0.000,C 90.000,E1 59.410} C_DIS
LIN {X 0.096,Y -592.442,Z 1241.123,A 0.000,B 0.000,C 90.000,E1 58.074} C_DIS
LIN {X -0.214,Y -593.498,Z 1241.117,A 0.000,B 0.000,C 90.000,E1 57.041} C_DIS
LIN {X -0.064,Y -594.911,Z 1241.108,A 0.000,B 0.000,C 90.000,E1 55.435} C_DIS
LIN {X 0.119,Y -596.270,Z 1241.099,A 0.000,B 0.000,C 90.000,E1 53.829} C_DIS
LIN {X -0.164,Y -597.447,Z 1241.090,A 0.000,B 0.000,C 90.000,E1 52.271} C_DIS
LIN {X 0.303,Y -598.315,Z 1241.084,A 0.000,B 0.000,C 90.000,E1 51.170} C_DIS
LIN {X -0.063,Y -598.883,Z 1241.079,A 0.000,B 0.000,C 90.000,E1 50.150} C_DIS
LIN {X -0.041,Y -599.417,Z 1241.073,A 0.000,B 0.000,C 90.000,E1 49.094} C_DIS
LIN {X -0.014,Y -599.850,Z 1241.067,A 0.000,B 0.000,C 90.000,E1 48.038} C_DIS
LIN {X 0.193,Y -600.156,Z 1241.063,A 0.000,B 0.000,C 90.000,E1 47.229} C_DIS
LIN {X -0.213,Y -600.360,Z 1241.057,A 0.000,B 0.000,C 90.000,E1 46.215} C_DIS
LIN {X 0.014,Y -600.463,Z 1241.049,A 0.000,B 0.000,C 90.000,E1 44.879} C_DIS
LIN {X 0.037,Y -600.314,Z 1241.044,A 0.000,B 0.000,C 90.000,E1 43.824} C_DIS
LIN {X -0.164,Y -599.968,Z 1241.036,A 0.000,B 0.000,C 90.000,E1 42.528} C_DIS
LIN {X -0.127,Y -599.493,Z 1241.030,A 0.000,B 0.000,C 90.000,E1 41.472} C_DIS
LIN {X -0.090,Y -598.923,Z 1241.025,A 0.000,B 0.000,C 90.000,E1 40.415} C_DIS
LIN {X -0.062,Y -598.399,Z 1241.019,A 0.000,B 0.000,C 90.000,E1 39.358} C_DIS
LIN {X -0.050,Y -597.571,Z 1241.013,A 0.000,B 0.000,C 90.000,E1 38.302} C_DIS
LIN {X 0.046,Y -596.546,Z 1241.007,A 0.000,B 0.000,C 90.000,E1 37.237} C_DIS
LIN {X -0.093,Y -595.641,Z 1241.003,A 0.000,B 0.000,C 90.000,E1 36.457} C_DIS
LIN {X 0.106,Y -594.540,Z 1240.998,A 0.000,B 0.000,C 90.000,E1 35.644} C_DIS
LIN {X -0.182,Y -592.823,Z 1240.992,A 0.000,B 0.000,C 90.000,E1 34.612} C_DIS
LIN {X 0.126,Y -591.317,Z 1240.988,A 0.000,B 0.000,C 90.000,E1 33.785} C_DIS
LIN {X -0.279,Y -590.220,Z 1240.985,A 0.000,B 0.000,C 90.000,E1 33.293} C_DIS
LIN {X -0.126,Y -587.462,Z 1240.979,A 0.000,B 0.000,C 90.000,E1 32.212} C_DIS
LIN {X 0.117,Y -585.114,Z 1240.974,A 0.000,B 0.000,C 90.000,E1 31.386} C_DIS
LIN {X 0.028,Y -582.348,Z 1240.970,A 0.000,B 0.000,C 90.000,E1 30.590} C_DIS
LIN {X 0.051,Y -580.281,Z 1240.967,A 0.000,B 0.000,C 90.000,E1 30.050} C_DIS
LIN {X -0.229,Y -578.034,Z 1240.964,A 0.000,B 0.000,C 90.000,E1 29.539} C_DIS
LIN {X 0.266,Y -575.569,Z 1240.961,A 0.000,B 0.000,C 90.000,E1 28.949} C_DIS
LIN {X -0.095,Y -569.995,Z 1240.955,A 0.000,B 0.000,C 90.000,E1 27.897} C_DIS
LIN {X -0.020,Y -566.069,Z 1240.951,A 0.000,B 0.000,C 90.000,E1 27.206} C_DIS
LIN {X 0.182,Y -560.955,Z 1240.947,A 0.000,B 0.000,C 90.000,E1 26.360} C_DIS
LIN {X -0.215,Y -557.265,Z 1240.943,A 0.000,B 0.000,C 90.000,E1 25.848} C_DIS
LIN {X 0.145,Y -551.285,Z 1240.939,A 0.000,B 0.000,C 90.000,E1 24.975} C_DIS
LIN {X -0.313,Y -546.929,Z 1240.936,A 0.000,B 0.000,C 90.000,E1 24.463} C_DIS
LIN {X -0.302,Y -542.332,Z 1240.933,A 0.000,B 0.000,C 90.000,E1 23.898} C_DIS
LIN {X 0.138,Y -532.355,Z 1240.926,A 0.000,B 0.000,C 90.000,E1 22.717} C_DIS
LIN {X -0.275,Y -528.453,Z 1240.924,A 0.000,B 0.000,C 90.000,E1 22.333} C_DIS
LIN {X -0.102,Y -519.312,Z 1240.919,A 0.000,B 0.000,C 90.000,E1 21.354} C_DIS
LIN {X 0.130,Y -508.588,Z 1240.913,A 0.000,B 0.000,C 90.000,E1 20.248} C_DIS
LIN {X -0.152,Y -498.796,Z 1240.907,A 0.000,B 0.000,C 90.000,E1 19.322} C_DIS
LIN {X -0.066,Y -487.206,Z 1240.901,A 0.000,B 0.000,C 90.000,E1 18.236} C_DIS
LIN {X -0.176,Y -479.720,Z 1240.898,A 0.000,B 0.000,C 90.000,E1 17.583} C_DIS
LIN {X -0.062,Y -464.933,Z 1240.890,A 0.000,B 0.000,C 90.000,E1 16.260} C_DIS
LIN {X 0.178,Y -445.753,Z 1240.881,A 0.000,B 0.000,C 90.000,E1 14.481} C_DIS
LIN {X 0.142,Y -425.404,Z 1240.870,A 0.000,B 0.000,C 90.000,E1 12.479} C_DIS
LIN {X -0.070,Y -402.741,Z 1240.856,A 0.000,B 0.000,C 90.000,E1 10.018} C_DIS
LIN {X -0.133,Y -400.240,Z 1240.854,A 0.000,B 0.000,C 90.000,E1 9.726} C_DIS
LIN {X 0.058,Y -395.853,Z 1240.851,A 0.000,B 0.000,C 90.000,E1 9.095} C_DIS
LIN {X 0.012,Y -394.339,Z 1240.849,A 0.000,B 0.000,C 90.000,E1 8.746} C_DIS
LIN {X -0.022,Y -394.335,Z 1240.849,A 0.000,B 0.000,C 90.000,E1 8.746} C_DIS
LIN {X -0.165,Y -394.261,Z 1240.848,A 0.000,B 0.000,C 90.000,E1 8.624} C_DIS
LIN {X 0.187,Y -394.259,Z 1240.848,A 0.000,B 0.000,C 90.000,E1 8.568} C_DIS
LIN {X -0.172,Y -396.519,Z 1240.845,A 0.000,B 0.000,C 90.000,E1 8.106} C_DIS
LIN {X -0.056,Y -399.672,Z 1240.843,A 0.000,B 0.000,C 90.000,E1 7.757} C_DIS
LIN {X 0.053,Y -401.333,Z 1240.842,A 0.000,B 0.000,C 90.000,E1 7.587} C_DIS
LIN {X -0.088,Y -407.027,Z 1240.840,A 0.000,B 0.000,C 90.000,E1 7.182} C_DIS
LIN {X 0.114,Y -413.278,Z 1240.838,A 0.000,B 0.000,C 90.000,E1 6.720} C_DIS
LIN {X 0.013,Y -421.390,Z 1240.834,A 0.000,B 0.000,C 90.000,E1 6.144} C_DIS
LIN {X -0.043,Y -430.795,Z 1240.830,A 0.000,B 0.000,C 90.000,E1 5.454} C_DIS
LIN {X -0.062,Y -443.311,Z 1240.825,A 0.000,B 0.000,C 90.000,E1 4.473} C_DIS
LIN {X -0.209,Y -455.773,Z 1240.819,A 0.000,B 0.000,C 90.000,E1 3.498} C_DIS
LIN {X -0.044,Y -461.937,Z 1240.817,A 0.000,B 0.000,C 90.000,E1 2.980} C_DIS
LIN {X -0.076,Y -469.459,Z 1240.813,A 0.000,B 0.000,C 90.000,E1 2.350} C_DIS
LIN {X 0.024,Y -473.843,Z 1240.811,A 0.000,B 0.000,C 90.000,E1 1.949} C_DIS
LIN {X 0.068,Y -478.219,Z 1240.809,A 0.000,B 0.000,C 90.000,E1 1.547} C_DIS
LIN {X 0.043,Y -485.060,Z 1240.805,A 0.000,B 0.000,C 90.000,E1 0.859} C_DIS
LIN {X 0.000,Y -492.802,Z 1240.800,A 0.000,B 0.000,C 90.000,E1 360.000} C_DIS
LIN {X 0.081,Y -497.169,Z 1240.797,A 0.000,B 0.000,C 90.000,E1 359.484} C_DIS
LIN {X 0.002,Y -503.038,Z 1240.793,A 0.000,B 0.000,C 90.000,E1 358.740} C_DIS
LIN {X -0.012,Y -508.412,Z 1240.789,A 0.000,B 0.000,C 90.000,E1 357.993} C_DIS
LIN {X 0.222,Y -514.359,Z 1240.784,A 0.000,B 0.000,C 90.000,E1 357.078} C_DIS
LIN {X 0.098,Y -518.125,Z 1240.781,A 0.000,B 0.000,C 90.000,E1 356.502} C_DIS
LIN {X 0.004,Y -521.653,Z 1240.777,A 0.000,B 0.000,C 90.000,E1 355.927} C_DIS
LIN {X 0.177,Y -525.622,Z 1240.773,A 0.000,B 0.000,C 90.000,E1 355.179} C_DIS
LIN {X -0.141,Y -529.250,Z 1240.769,A 0.000,B 0.000,C 90.000,E1 354.489} C_DIS
LIN {X -0.152,Y -531.968,Z 1240.766,A 0.000,B 0.000,C 90.000,E1 353.913} C_DIS
LIN {X -0.145,Y -534.517,Z 1240.763,A 0.000,B 0.000,C 90.000,E1 353.337} C_DIS
LIN {X -0.122,Y -536.889,Z 1240.760,A 0.000,B 0.000,C 90.000,E1 352.761} C_DIS
LIN {X -0.024,Y -540.093,Z 1240.755,A 0.000,B 0.000,C 90.000,E1 351.894} C_DIS
LIN {X 0.106,Y -543.024,Z 1240.750,A 0.000,B 0.000,C 90.000,E1 351.027} C_DIS
LIN {X -0.182,Y -545.773,Z 1240.745,A 0.000,B 0.000,C 90.000,E1 350.208} C_DIS
LIN {X 0.104,Y -548.976,Z 1240.739,A 0.000,B 0.000,C 90.000,E1 349.050} C_DIS
LIN {X 0.112,Y -552.558,Z 1240.731,A 0.000,B 0.000,C 90.000,E1 347.645} C_DIS
LIN {X 0.306,Y -555.693,Z 1240.724,A 0.000,B 0.000,C 90.000,E1 346.228} C_DIS
LIN {X 0.022,Y -558.372,Z 1240.716,A 0.000,B 0.000,C 90.000,E1 344.866} C_DIS
LIN {X 0.040,Y -559.854,Z 1240.711,A 0.000,B 0.000,C 90.000,E1 344.031} C_DIS
LIN {X 0.075,Y -561.215,Z 1240.707,A 0.000,B 0.000,C 90.000,E1 343.196} C_DIS
LIN {X 0.033,Y -563.054,Z 1240.699,A 0.000,B 0.000,C 90.000,E1 341.819} C_DIS
LIN {X -0.125,Y -564.219,Z 1240.693,A 0.000,B 0.000,C 90.000,E1 340.732} C_DIS
LIN {X -0.077,Y -564.970,Z 1240.687,A 0.000,B 0.000,C 90.000,E1 339.625} C_DIS
LIN {X 0.184,Y -565.263,Z 1240.682,A 0.000,B 0.000,C 90.000,E1 338.773} C_DIS
LIN {X 0.111,Y -565.268,Z 1240.679,A 0.000,B 0.000,C 90.000,E1 338.230} C_DIS
LIN {X 0.054,Y -565.008,Z 1240.675,A 0.000,B 0.000,C 90.000,E1 337.411} C_DIS
LIN {X -0.028,Y -564.657,Z 1240.672,A 0.000,B 0.000,C 90.000,E1 336.869} C_DIS
LIN {X -0.278,Y -563.460,Z 1240.665,A 0.000,B 0.000,C 90.000,E1 335.793} C_DIS
LIN {X -0.149,Y -562.693,Z 1240.662,A 0.000,B 0.000,C 90.000,E1 335.229} C_DIS
LIN {X 0.083,Y -560.613,Z 1240.656,A 0.000,B 0.000,C 90.000,E1 334.101} C_DIS
LIN {X 0.024,Y -558.087,Z 1240.650,A 0.000,B 0.000,C 90.000,E1 332.999} C_DIS
LIN {X 0.150,Y -555.499,Z 1240.645,A 0.000,B 0.000,C 90.000,E1 332.153} C_DIS
LIN {X -0.281,Y -553.707,Z 1240.642,A 0.000,B 0.000,C 90.000,E1 331.641} C_DIS
LIN {X -0.201,Y -550.309,Z 1240.638,A 0.000,B 0.000,C 90.000,E1 330.795} C_DIS
LIN {X 0.106,Y -546.271,Z 1240.633,A 0.000,B 0.000,C 90.000,E1 329.921} C_DIS
LIN {X 0.220,Y -542.397,Z 1240.629,A 0.000,B 0.000,C 90.000,E1 329.203} C_DIS
LIN {X -0.024,Y -536.984,Z 1240.624,A 0.000,B 0.000,C 90.000,E1 328.377} C_DIS
LIN {X -0.148,Y -531.172,Z 1240.620,A 0.000,B 0.000,C 90.000,E1 327.533} C_DIS
LIN {X 0.226,Y -524.906,Z 1240.615,A 0.000,B 0.000,C 90.000,E1 326.628} C_DIS
LIN {X -0.157,Y -517.613,Z 1240.609,A 0.000,B 0.000,C 90.000,E1 325.674} C_DIS
LIN {X 0.011,Y -513.932,Z 1240.606,A 0.000,B 0.000,C 90.000,E1 325.102} C_DIS
LIN {X 0.185,Y -510.990,Z 1240.603,A 0.000,B 0.000,C 90.000,E1 324.562} C_DIS
LIN {X 0.144,Y -508.787,Z 1240.601,A 0.000,B 0.000,C 90.000,E1 324.069} C_DIS
LIN {X -0.016,Y -507.227,Z 1240.597,A 0.000,B 0.000,C 90.000,E1 323.497} C_DIS
LIN {X -0.209,Y -506.087,Z 1240.594,A 0.000,B 0.000,C 90.000,E1 322.924} C_DIS
LIN {X 0.193,Y -505.150,Z 1240.589,A 0.000,B 0.000,C 90.000,E1 321.984} C_DIS
LIN {X 0.190,Y -504.958,Z 1240.584,A 0.000,B 0.000,C 90.000,E1 321.090} C_DIS
LIN {X 0.188,Y -505.667,Z 1240.574,A 0.000,B 0.000,C 90.000,E1 319.299} C_DIS
LIN {X -0.073,Y -506.250,Z 1240.566,A 0.000,B 0.000,C 90.000,E1 317.838} C_DIS
LIN {X -0.095,Y -506.870,Z 1240.556,A 0.000,B 0.000,C 90.000,E1 316.053} C_DIS
LIN {X 0.113,Y -507.431,Z 1240.544,A 0.000,B 0.000,C 90.000,E1 313.947} C_DIS
LIN {X -0.027,Y -508.149,Z 1240.533,A 0.000,B 0.000,C 90.000,E1 311.881} C_DIS
LIN {X -0.101,Y -508.590,Z 1240.526,A 0.000,B 0.000,C 90.000,E1 310.701} C_DIS
LIN {X 0.072,Y -508.996,Z 1240.518,A 0.000,B 0.000,C 90.000,E1 309.197} C_DIS
LIN {X -0.165,Y -509.527,Z 1240.508,A 0.000,B 0.000,C 90.000,E1 307.443} C_DIS
LIN {X 0.188,Y -509.843,Z 1240.501,A 0.000,B 0.000,C 90.000,E1 306.217} C_DIS
LIN {X 0.155,Y -510.145,Z 1240.493,A 0.000,B 0.000,C 90.000,E1 304.739} C_DIS
LIN {X -0.163,Y -510.426,Z 1240.485,A 0.000,B 0.000,C 90.000,E1 303.293} C_DIS
LIN {X 0.290,Y -510.592,Z 1240.475,A 0.000,B 0.000,C 90.000,E1 301.465} C_DIS
LIN {X -0.215,Y -510.649,Z 1240.465,A 0.000,B 0.000,C 90.000,E1 299.745} C_DIS
LIN {X -0.008,Y -510.631,Z 1240.459,A 0.000,B 0.000,C 90.000,E1 298.537} C_DIS
LIN {X 0.036,Y -510.567,Z 1240.450,A 0.000,B 0.000,C 90.000,E1 297.052} C_DIS
LIN {X 0.138,Y -510.711,Z 1240.434,A 0.000,B 0.000,C 90.000,E1 294.079} C_DIS
LIN {X 0.110,Y -510.714,Z 1240.427,A 0.000,B 0.000,C 90.000,E1 292.898} C_DIS
LIN {X 0.084,Y -510.372,Z 1240.421,A 0.000,B 0.000,C 90.000,E1 291.716} C_DIS
LIN {X -0.029,Y -509.740,Z 1240.412,A 0.000,B 0.000,C 90.000,E1 290.248} C_DIS
LIN {X -0.055,Y -508.969,Z 1240.403,A 0.000,B 0.000,C 90.000,E1 288.471} C_DIS
LIN {X -0.036,Y -508.393,Z 1240.394,A 0.000,B 0.000,C 90.000,E1 286.985} C_DIS
LIN {X 0.040,Y -507.902,Z 1240.388,A 0.000,B 0.000,C 90.000,E1 285.788} C_DIS
LIN {X 0.101,Y -507.326,Z 1240.381,A 0.000,B 0.000,C 90.000,E1 284.592} C_DIS
LIN {X 0.019,Y -506.581,Z 1240.375,A 0.000,B 0.000,C 90.000,E1 283.411} C_DIS
LIN {X -0.185,Y -505.734,Z 1240.368,A 0.000,B 0.000,C 90.000,E1 282.243} C_DIS
LIN {X 0.253,Y -505.084,Z 1240.363,A 0.000,B 0.000,C 90.000,E1 281.299} C_DIS
LIN {X -0.242,Y -503.525,Z 1240.351,A 0.000,B 0.000,C 90.000,E1 279.265} C_DIS
LIN {X 0.152,Y -502.219,Z 1240.340,A 0.000,B 0.000,C 90.000,E1 277.125} C_DIS
LIN {X 0.082,Y -501.255,Z 1240.330,A 0.000,B 0.000,C 90.000,E1 275.334} C_DIS
LIN {X 0.240,Y -500.739,Z 1240.325,A 0.000,B 0.000,C 90.000,E1 274.416} C_DIS
LIN {X 0.043,Y -499.729,Z 1240.315,A 0.000,B 0.000,C 90.000,E1 272.636} C_DIS
LIN {X -0.073,Y -498.572,Z 1240.306,A 0.000,B 0.000,C 90.000,E1 271.146} C_DIS
LIN {X -0.121,Y -496.891,Z 1240.293,A 0.000,B 0.000,C 90.000,E1 268.740} C_DIS
LIN {X 0.065,Y -495.812,Z 1240.283,A 0.000,B 0.000,C 90.000,E1 266.906} C_DIS
LIN {X -0.206,Y -494.803,Z 1240.273,A 0.000,B 0.000,C 90.000,E1 265.122} C_DIS
LIN {X -0.225,Y -494.007,Z 1240.266,A 0.000,B 0.000,C 90.000,E1 263.913} C_DIS
LIN {X 0.125,Y -492.894,Z 1240.258,A 0.000,B 0.000,C 90.000,E1 262.356} C_DIS
LIN {X 0.234,Y -492.048,Z 1240.253,A 0.000,B 0.000,C 90.000,E1 261.432} C_DIS
LIN {X -0.104,Y -489.981,Z 1240.241,A 0.000,B 0.000,C 90.000,E1 259.342} C_DIS
LIN {X 0.059,Y -488.094,Z 1240.227,A 0.000,B 0.000,C 90.000,E1 256.881} C_DIS
LIN {X -0.071,Y -486.570,Z 1240.214,A 0.000,B 0.000,C 90.000,E1 254.448} C_DIS
LIN {X 0.020,Y -485.465,Z 1240.203,A 0.000,B 0.000,C 90.000,E1 252.598} C_DIS
LIN {X 0.225,Y -484.502,Z 1240.193,A 0.000,B 0.000,C 90.000,E1 250.732} C_DIS
LIN {X 0.100,Y -483.746,Z 1240.185,A 0.000,B 0.000,C 90.000,E1 249.209} C_DIS
LIN {X 0.132,Y -482.955,Z 1240.176,A 0.000,B 0.000,C 90.000,E1 247.667} C_DIS
LIN {X -0.103,Y -481.782,Z 1240.166,A 0.000,B 0.000,C 90.000,E1 245.845} C_DIS
LIN {X 0.077,Y -480.629,Z 1240.157,A 0.000,B 0.000,C 90.000,E1 244.280} C_DIS
LIN {X 0.005,Y -479.468,Z 1240.149,A 0.000,B 0.000,C 90.000,E1 242.743} C_DIS
LIN {X 0.132,Y -478.182,Z 1240.140,A 0.000,B 0.000,C 90.000,E1 241.179} C_DIS
LIN {X -0.183,Y -476.817,Z 1240.131,A 0.000,B 0.000,C 90.000,E1 239.665} C_DIS
LIN {X -0.121,Y -474.407,Z 1240.118,A 0.000,B 0.000,C 90.000,E1 237.168} C_DIS
LIN {X -0.110,Y -471.868,Z 1240.102,A 0.000,B 0.000,C 90.000,E1 234.356} C_DIS
LIN {X 0.032,Y -470.141,Z 1240.090,A 0.000,B 0.000,C 90.000,E1 232.145} C_DIS
LIN {X -0.020,Y -468.267,Z 1240.078,A 0.000,B 0.000,C 90.000,E1 229.952} C_DIS
LIN {X -0.240,Y -467.036,Z 1240.069,A 0.000,B 0.000,C 90.000,E1 228.405} C_DIS
LIN {X 0.126,Y -465.868,Z 1240.060,A 0.000,B 0.000,C 90.000,E1 226.782} C_DIS
LIN {X 0.014,Y -463.708,Z 1240.035,A 0.000,B 0.000,C 90.000,E1 222.366} C_DIS
LIN {X -0.093,Y -464.952,Z 1239.998,A 0.000,B 0.000,C 90.000,E1 215.724} C_DIS
LIN {X 0.265,Y -468.228,Z 1239.974,A 0.000,B 0.000,C 90.000,E1 211.258} C_DIS
LIN {X 0.067,Y -472.366,Z 1239.953,A 0.000,B 0.000,C 90.000,E1 207.513} C_DIS
LIN {X -0.186,Y -474.731,Z 1239.943,A 0.000,B 0.000,C 90.000,E1 205.668} C_DIS
LIN {X 0.156,Y -479.646,Z 1239.923,A 0.000,B 0.000,C 90.000,E1 202.206} C_DIS
LIN {X -0.037,Y -485.119,Z 1239.906,A 0.000,B 0.000,C 90.000,E1 199.141} C_DIS
LIN {X -0.026,Y -491.716,Z 1239.889,A 0.000,B 0.000,C 90.000,E1 196.079} C_DIS
LIN {X 0.276,Y -494.577,Z 1239.883,A 0.000,B 0.000,C 90.000,E1 194.828} C_DIS
LIN {X -0.238,Y -499.687,Z 1239.871,A 0.000,B 0.000,C 90.000,E1 192.771} C_DIS
LIN {X -0.194,Y -505.692,Z 1239.858,A 0.000,B 0.000,C 90.000,E1 190.366} C_DIS
LIN {X -0.126,Y -511.228,Z 1239.846,A 0.000,B 0.000,C 90.000,E1 188.276} C_DIS
LIN {X 0.065,Y -515.197,Z 1239.838,A 0.000,B 0.000,C 90.000,E1 186.777} C_DIS
LIN {X -0.181,Y -519.050,Z 1239.830,A 0.000,B 0.000,C 90.000,E1 185.334} C_DIS
LIN {X 0.059,Y -523.718,Z 1239.820,A 0.000,B 0.000,C 90.000,E1 183.555} C_DIS
LIN {X -0.142,Y -528.291,Z 1239.810,A 0.000,B 0.000,C 90.000,E1 181.835} C_DIS
LIN {X -0.217,Y -531.290,Z 1239.804,A 0.000,B 0.000,C 90.000,E1 180.688} C_DIS
LIN {X -0.262,Y -534.290,Z 1239.797,A 0.000,B 0.000,C 90.000,E1 179.542} C_DIS
LIN {X -0.245,Y -537.902,Z 1239.789,A 0.000,B 0.000,C 90.000,E1 178.108} C_DIS
